LIN {X 0,Y 228.351,Z 344.664,A -85,B 0,C 180,E1 -20167.071,E2 -20167.071} C_VEL
LIN {X 0,Y 228.165,Z 344.686,A -85,B 0,C 180,E1 -20170.65,E2 -20170.65} C_VEL
LIN {X 0,Y 228.051,Z 344.704,A -85,B 0,C 180,E1 -20176.102,E2 -20176.102} C_VEL
LIN {X 0,Y 227.936,Z 344.714,A -85,B 0,C 180,E1 -20179.826,E2 -20179.826} C_VEL
LIN {X 0,Y 227.907,Z 344.72,A -85,B 0,C 180,E1 -20183.633,E2 -20183.633} C_VEL
LIN {X 0,Y 227.879,Z 344.721,A -85,B 0,C 180,E1 -20187.556,E2 -20187.556} C_VEL
LIN {X 0,Y 227.867,Z 344.726,A -85,B 0,C 180,E1 -20191.622,E2 -20191.622} C_VEL
LIN {X 0,Y 227.974,Z 344.855,A -85,B 0,C 180,E1 -20194.37,E2 -20194.37} C_VEL
LIN {X 0,Y 229.283,Z 351.773,A -85,B 0,C 180,E1 -20198.929,E2 -20198.929} C_VEL
LIN {X 0,Y 231.078,Z 360.512,A -85,B 0,C 180,E1 -20204.388,E2 -20204.388} C_VEL
LIN {X 0,Y 232.42,Z 367.069,A -85,B 0,C 180,E1 -20208.302,E2 -20208.302} C_VEL
LIN {X 0,Y 231.376,Z 372.602,A -85,B 0,C 180,E1 -20211.43,E2 -20211.43} C_VEL
LIN {X 0,Y 229.532,Z 381.682,A -85,B 0,C 180,E1 -20216.557,E2 -20216.557} C_VEL
LIN {X 0,Y 228.619,Z 387.309,A -85,B 0,C 180,E1 -20219.581,E2 -20219.581} C_VEL
LIN {X 0,Y 229.454,Z 407.428,A -85,B 0,C 180,E1 -20221.235,E2 -20221.235} C_VEL
LIN {X 0,Y 229.647,Z 410.827,A -85,B 0,C 180,E1 -20221.565,E2 -20221.565} C_VEL
LIN {X 0,Y 229.388,Z 416.398,A -85,B 0,C 180,E1 -20222.127,E2 -20222.127} C_VEL
LIN {X 0,Y 226.978,Z 425.249,A -85,B 0,C 180,E1 -20223.098,E2 -20223.098} C_VEL
LIN {X 0,Y 224.51,Z 433.801,A -85,B 0,C 180,E1 -20224.199,E2 -20224.199} C_VEL
LIN {X 0,Y 224.14,Z 438.823,A -85,B 0,C 180,E1 -20224.956,E2 -20224.956} C_VEL
LIN {X 0,Y 225.046,Z 452.21,A -85,B 0,C 180,E1 -20227.268,E2 -20227.268} C_VEL
LIN {X 0,Y 225.004,Z 455.94,A -85,B 0,C 180,E1 -20227.989,E2 -20227.989} C_VEL
LIN {X 0,Y 223.355,Z 467.739,A -85,B 0,C 180,E1 -20230.632,E2 -20230.632} C_VEL
LIN {X 0,Y 221.995,Z 477.991,A -85,B 0,C 180,E1 -20233.447,E2 -20233.447} C_VEL
LIN {X 0,Y 221.257,Z 486.356,A -85,B 0,C 180,E1 -20236.22,E2 -20236.22} C_VEL
LIN {X 0,Y 221.057,Z 493.355,A -85,B 0,C 180,E1 -20239.005,E2 -20239.005} C_VEL
LIN {X 0,Y 221.203,Z 499.088,A -85,B 0,C 180,E1 -20241.782,E2 -20241.782} C_VEL
LIN {X 0,Y 221.557,Z 503.69,A -85,B 0,C 180,E1 -20244.541,E2 -20244.541} C_VEL
LIN {X 0,Y 221.876,Z 506.14,A -85,B 0,C 180,E1 -20246.37,E2 -20246.37} C_VEL
LIN {X 0,Y 222.107,Z 508.099,A -85,B 0,C 180,E1 -20248.188,E2 -20248.188} C_VEL
LIN {X 0,Y 222.354,Z 509.63,A -85,B 0,C 180,E1 -20250.002,E2 -20250.002} C_VEL
LIN {X 0,Y 221.73,Z 510.553,A -85,B 0,C 180,E1 -20251.818,E2 -20251.818} C_VEL
LIN {X 0,Y 220.533,Z 511.308,A -85,B 0,C 180,E1 -20255.488,E2 -20255.488} C_VEL
LIN {X 0,Y 219.744,Z 510.766,A -85,B 0,C 180,E1 -20259.203,E2 -20259.203} C_VEL
LIN {X 0,Y 219.781,Z 509.022,A -85,B 0,C 180,E1 -20262.936,E2 -20262.936} C_VEL
LIN {X 0,Y 220.864,Z 506.171,A -85,B 0,C 180,E1 -20266.643,E2 -20266.643} C_VEL
LIN {X 0,Y 223.015,Z 502.256,A -85,B 0,C 180,E1 -20270.284,E2 -20270.284} C_VEL
LIN {X 0,Y 226.28,Z 497.299,A -85,B 0,C 180,E1 -20273.815,E2 -20273.815} C_VEL
LIN {X 0,Y 232.087,Z 489.566,A -85,B 0,C 180,E1 -20277.995,E2 -20277.995} C_VEL
LIN {X 0,Y 237.04,Z 483.14,A -85,B 0,C 180,E1 -20280.762,E2 -20280.762} C_VEL
LIN {X 0,Y 242.014,Z 476.891,A -85,B 0,C 180,E1 -20282.992,E2 -20282.992} C_VEL
LIN {X 0,Y 249.318,Z 466.525,A -85,B 0,C 180,E1 -20286.298,E2 -20286.298} C_VEL
LIN {X 0,Y 253.481,Z 460.309,A -85,B 0,C 180,E1 -20288.092,E2 -20288.092} C_VEL
LIN {X 0,Y 258.603,Z 451.554,A -85,B 0,C 180,E1 -20290.712,E2 -20290.712} C_VEL
LIN {X 0,Y 262.82,Z 443.829,A -85,B 0,C 180,E1 -20293.242,E2 -20293.242} C_VEL
LIN {X 0,Y 267.388,Z 435.806,A -85,B 0,C 180,E1 -20296.26,E2 -20296.26} C_VEL
LIN {X 0,Y 268.712,Z 433.696,A -85,B 0,C 180,E1 -20297.156,E2 -20297.156} C_VEL
LIN {X 0,Y 269.675,Z 431.962,A -85,B 0,C 180,E1 -20298.28,E2 -20298.28} C_VEL
LIN {X 0,Y 270.402,Z 430.463,A -85,B 0,C 180,E1 -20301.407,E2 -20301.407} C_VEL
LIN {X 0,Y 270.864,Z 430.408,A -85,B 0,C 180,E1 -20303.549,E2 -20303.549} C_VEL
LIN {X 0,Y 270.034,Z 431.543,A -85,B 0,C 180,E1 -20304.344,E2 -20304.344} C_VEL
LIN {X 0,Y 260.6,Z 440.793,A -85,B 0,C 180,E1 -20307.36,E2 -20307.36} C_VEL
LIN {X 0,Y 253.365,Z 447.035,A -85,B 0,C 180,E1 -20310.047,E2 -20310.047} C_VEL
LIN {X 0,Y 246.809,Z 451.946,A -85,B 0,C 180,E1 -20312.896,E2 -20312.896} C_VEL
LIN {X 0,Y 241.057,Z 455.609,A -85,B 0,C 180,E1 -20315.91,E2 -20315.91} C_VEL
LIN {X 0,Y 235.987,Z 458.133,A -85,B 0,C 180,E1 -20319.061,E2 -20319.061} C_VEL
LIN {X 0,Y 231.716,Z 459.508,A -85,B 0,C 180,E1 -20322.344,E2 -20322.344} C_VEL
LIN {X 0,Y 228.11,Z 459.778,A -85,B 0,C 180,E1 -20325.731,E2 -20325.731} C_VEL
LIN {X 0,Y 225.275,Z 458.892,A -85,B 0,C 180,E1 -20329.212,E2 -20329.212} C_VEL
LIN {X 0,Y 223.148,Z 456.815,A -85,B 0,C 180,E1 -20332.763,E2 -20332.763} C_VEL
LIN {X 0,Y 221.835,Z 453.504,A -85,B 0,C 180,E1 -20336.368,E2 -20336.368} C_VEL
LIN {X 0,Y 221.174,Z 448.92,A -85,B 0,C 180,E1 -20340,E2 -20340} C_VEL
LIN {X 0,Y 220.811,Z 442.957,A -85,B 0,C 180,E1 -20343.65,E2 -20343.65} C_VEL
LIN {X 0,Y 221.237,Z 435.436,A -85,B 0,C 180,E1 -20347.301,E2 -20347.301} C_VEL
LIN {X 0,Y 222.005,Z 427.386,A -85,B 0,C 180,E1 -20350.488,E2 -20350.488} C_VEL
LIN {X 0,Y 223.089,Z 417.659,A -85,B 0,C 180,E1 -20353.667,E2 -20353.667} C_VEL
LIN {X 0,Y 224.375,Z 407.773,A -85,B 0,C 180,E1 -20356.374,E2 -20356.374} C_VEL
LIN {X 0,Y 226.11,Z 394.99,A -85,B 0,C 180,E1 -20359.284,E2 -20359.284} C_VEL
LIN {X 0,Y 228.029,Z 382.007,A -85,B 0,C 180,E1 -20361.707,E2 -20361.707} C_VEL
LIN {X 0,Y 228.741,Z 375.181,A -85,B 0,C 180,E1 -20362.815,E2 -20362.815} C_VEL
LIN {X 0,Y 224.992,Z 361.192,A -85,B 0,C 180,E1 -20365.058,E2 -20365.058} C_VEL
LIN {X 0,Y 220.994,Z 346.136,A -85,B 0,C 180,E1 -20367.173,E2 -20367.173} C_VEL
LIN {X 0,Y 220.946,Z 345.626,A -85,B 0,C 180,E1 -20367.474,E2 -20367.474} C_VEL
LIN {X 0,Y 220.869,Z 345.599,A -85,B 0,C 180,E1 -20370.778,E2 -20370.778} C_VEL
LIN {X 0,Y 220.807,Z 345.604,A -85,B 0,C 180,E1 -20374.955,E2 -20374.955} C_VEL
LIN {X 0,Y 220.812,Z 345.602,A -85,B 0,C 180,E1 -20379.536,E2 -20379.536} C_VEL
LIN {X 0,Y 220.781,Z 345.607,A -85,B 0,C 180,E1 -20384.453,E2 -20384.453} C_VEL
LIN {X 0,Y 220.809,Z 345.604,A -85,B 0,C 180,E1 -20388.055,E2 -20388.055} C_VEL
LIN {X 0,Y 220.84,Z 345.597,A -85,B 0,C 180,E1 -20392.794,E2 -20392.794} C_VEL
LIN {X 0,Y 220.829,Z 345.601,A -85,B 0,C 180,E1 -20397.244,E2 -20397.244} C_VEL
LIN {X 0,Y 220.833,Z 345.598,A -85,B 0,C 180,E1 -20401.484,E2 -20401.484} C_VEL
LIN {X 0,Y 220.868,Z 345.596,A -85,B 0,C 180,E1 -20405.563,E2 -20405.563} C_VEL
LIN {X 0,Y 220.891,Z 345.592,A -85,B 0,C 180,E1 -20409.512,E2 -20409.512} C_VEL
LIN {X 0,Y 221.022,Z 345.576,A -85,B 0,C 180,E1 -20413.369,E2 -20413.369} C_VEL
LIN {X 0,Y 221.122,Z 345.561,A -85,B 0,C 180,E1 -20419.005,E2 -20419.005} C_VEL
LIN {X 0,Y 221.316,Z 345.54,A -85,B 0,C 180,E1 -20422.701,E2 -20422.701} C_VEL
LIN {X 0,Y 221.517,Z 345.514,A -85,B 0,C 180,E1 -20428.18,E2 -20428.18} C_VEL
LIN {X 0,Y 221.517,Z 345.518,A -85,B 0,C 180,E1 -20431.816,E2 -20431.816} C_VEL
LIN {X 0,Y 221.315,Z 345.539,A -85,B 0,C 180,E1 -20437.296,E2 -20437.296} C_VEL
LIN {X 0,Y 221.12,Z 345.565,A -85,B 0,C 180,E1 -20440.992,E2 -20440.992} C_VEL
LIN {X 0,Y 221.019,Z 345.576,A -85,B 0,C 180,E1 -20446.628,E2 -20446.628} C_VEL
LIN {X 0,Y 220.894,Z 345.592,A -85,B 0,C 180,E1 -20450.484,E2 -20450.484} C_VEL
LIN {X 0,Y 220.868,Z 345.593,A -85,B 0,C 180,E1 -20454.433,E2 -20454.433} C_VEL
LIN {X 0,Y 220.827,Z 345.601,A -85,B 0,C 180,E1 -20458.513,E2 -20458.513} C_VEL
LIN {X 0,Y 220.815,Z 345.6,A -85,B 0,C 180,E1 -20462.754,E2 -20462.754} C_VEL
LIN {X 0,Y 220.808,Z 345.606,A -85,B 0,C 180,E1 -20467.276,E2 -20467.276} C_VEL
LIN {X 0,Y 220.768,Z 345.607,A -85,B 0,C 180,E1 -20471.95,E2 -20471.95} C_VEL
LIN {X 0,Y 220.772,Z 345.609,A -85,B 0,C 180,E1 -20475.545,E2 -20475.545} C_VEL
LIN {X 0,Y 220.803,Z 345.602,A -85,B 0,C 180,E1 -20480.461,E2 -20480.461} C_VEL
LIN {X 0,Y 220.796,Z 345.607,A -85,B 0,C 180,E1 -20485.043,E2 -20485.043} C_VEL
LIN {X 0,Y 220.863,Z 345.596,A -85,B 0,C 180,E1 -20489.393,E2 -20489.393} C_VEL
LIN {X 0,Y 220.89,Z 345.593,A -85,B 0,C 180,E1 -20493.548,E2 -20493.548} C_VEL
LIN {X 0,Y 220.872,Z 345.594,A -85,B 0,C 180,E1 -20497.552,E2 -20497.552} C_VEL
LIN {X 0,Y 220.978,Z 345.585,A -85,B 0,C 180,E1 -20502.57,E2 -20502.57} C_VEL
LIN {X 0,Y 221.02,Z 345.577,A -85,B 0,C 180,E1 -20507.138,E2 -20507.138} C_VEL
LIN {X 0,Y 221.252,Z 345.549,A -85,B 0,C 180,E1 -20510.861,E2 -20510.861} C_VEL
LIN {X 0,Y 221.305,Z 345.54,A -85,B 0,C 180,E1 -20512.702,E2 -20512.702} C_VEL
LIN {X 0,Y 221.507,Z 345.519,A -85,B 0,C 180,E1 -20518.181,E2 -20518.181} C_VEL
LIN {X 0,Y 221.507,Z 345.514,A -85,B 0,C 180,E1 -20521.818,E2 -20521.818} C_VEL
LIN {X 0,Y 221.304,Z 345.541,A -85,B 0,C 180,E1 -20527.297,E2 -20527.297} C_VEL
LIN {X 0,Y 221.11,Z 345.563,A -85,B 0,C 180,E1 -20530.994,E2 -20530.994} C_VEL
LIN {X 0,Y 221.01,Z 345.578,A -85,B 0,C 180,E1 -20536.63,E2 -20536.63} C_VEL
LIN {X 0,Y 220.886,Z 345.594,A -85,B 0,C 180,E1 -20540.486,E2 -20540.486} C_VEL
LIN {X 0,Y 220.86,Z 345.598,A -85,B 0,C 180,E1 -20544.435,E2 -20544.435} C_VEL
LIN {X 0,Y 220.829,Z 345.6,A -85,B 0,C 180,E1 -20548.514,E2 -20548.514} C_VEL
LIN {X 0,Y 220.837,Z 345.602,A -85,B 0,C 180,E1 -20552.752,E2 -20552.752} C_VEL
LIN {X 0,Y 220.932,Z 345.761,A -85,B 0,C 180,E1 -20554.204,E2 -20554.204} C_VEL
LIN {X 0,Y 222.336,Z 353.162,A -85,B 0,C 180,E1 -20559.212,E2 -20559.212} C_VEL
LIN {X 0,Y 223.801,Z 360.205,A -85,B 0,C 180,E1 -20563.761,E2 -20563.761} C_VEL
LIN {X 0,Y 225.071,Z 366.093,A -85,B 0,C 180,E1 -20567.402,E2 -20567.402} C_VEL
LIN {X 0,Y 225.155,Z 368.839,A -85,B 0,C 180,E1 -20569.045,E2 -20569.045} C_VEL
LIN {X 0,Y 223.522,Z 376.147,A -85,B 0,C 180,E1 -20573.318,E2 -20573.318} C_VEL
LIN {X 0,Y 221.784,Z 385.568,A -85,B 0,C 180,E1 -20578.824,E2 -20578.824} C_VEL
LIN {X 0,Y 221.637,Z 386.569,A -85,B 0,C 180,E1 -20579.183,E2 -20579.183} C_VEL
LIN {X 0,Y 222.275,Z 404.267,A -85,B 0,C 180,E1 -20580.656,E2 -20580.656} C_VEL
LIN {X 0,Y 223.092,Z 419.696,A -85,B 0,C 180,E1 -20582.314,E2 -20582.314} C_VEL
LIN {X 0,Y 223.769,Z 433.244,A -85,B 0,C 180,E1 -20584.107,E2 -20584.107} C_VEL
LIN {X 0,Y 224.14,Z 438.823,A -85,B 0,C 180,E1 -20584.956,E2 -20584.956} C_VEL
LIN {X 0,Y 223.745,Z 443.842,A -85,B 0,C 180,E1 -20585.768,E2 -20585.768} C_VEL
LIN {X 0,Y 222.288,Z 448.619,A -85,B 0,C 180,E1 -20586.612,E2 -20586.612} C_VEL
LIN {X 0,Y 218.377,Z 457.615,A -85,B 0,C 180,E1 -20588.445,E2 -20588.445} C_VEL
LIN {X 0,Y 216.763,Z 463.504,A -85,B 0,C 180,E1 -20589.815,E2 -20589.815} C_VEL
LIN {X 0,Y 215.405,Z 473.343,A -85,B 0,C 180,E1 -20592.436,E2 -20592.436} C_VEL
LIN {X 0,Y 214.541,Z 482.269,A -85,B 0,C 180,E1 -20595.295,E2 -20595.295} C_VEL
LIN {X 0,Y 214.11,Z 490.839,A -85,B 0,C 180,E1 -20598.643,E2 -20598.643} C_VEL
LIN {X 0,Y 214.234,Z 496.795,A -85,B 0,C 180,E1 -20601.513,E2 -20601.513} C_VEL
LIN {X 0,Y 214.615,Z 501.559,A -85,B 0,C 180,E1 -20604.364,E2 -20604.364} C_VEL
LIN {X 0,Y 215.06,Z 505.244,A -85,B 0,C 180,E1 -20607.192,E2 -20607.192} C_VEL
LIN {X 0,Y 215.447,Z 507.895,A -85,B 0,C 180,E1 -20610.002,E2 -20610.002} C_VEL
LIN {X 0,Y 214.794,Z 508.897,A -85,B 0,C 180,E1 -20611.877,E2 -20611.877} C_VEL
LIN {X 0,Y 213.518,Z 509.799,A -85,B 0,C 180,E1 -20615.669,E2 -20615.669} C_VEL
LIN {X 0,Y 212.721,Z 509.42,A -85,B 0,C 180,E1 -20619.51,E2 -20619.51} C_VEL
LIN {X 0,Y 212.816,Z 507.904,A -85,B 0,C 180,E1 -20623.367,E2 -20623.367} C_VEL
LIN {X 0,Y 214.004,Z 505.324,A -85,B 0,C 180,E1 -20627.193,E2 -20627.193} C_VEL
LIN {X 0,Y 216.31,Z 501.701,A -85,B 0,C 180,E1 -20630.942,E2 -20630.942} C_VEL
LIN {X 0,Y 219.763,Z 497.027,A -85,B 0,C 180,E1 -20634.567,E2 -20634.567} C_VEL
LIN {X 0,Y 225.822,Z 489.776,A -85,B 0,C 180,E1 -20638.843,E2 -20638.843} C_VEL
LIN {X 0,Y 230.142,Z 484.601,A -85,B 0,C 180,E1 -20641.276,E2 -20641.276} C_VEL
LIN {X 0,Y 236.156,Z 477.821,A -85,B 0,C 180,E1 -20643.919,E2 -20643.919} C_VEL
LIN {X 0,Y 243.775,Z 468.048,A -85,B 0,C 180,E1 -20647.261,E2 -20647.261} C_VEL
LIN {X 0,Y 248.127,Z 462.176,A -85,B 0,C 180,E1 -20649.067,E2 -20649.067} C_VEL
LIN {X 0,Y 253.567,Z 453.945,A -85,B 0,C 180,E1 -20651.699,E2 -20651.699} C_VEL
LIN {X 0,Y 258.074,Z 446.707,A -85,B 0,C 180,E1 -20654.242,E2 -20654.242} C_VEL
LIN {X 0,Y 263.047,Z 439.181,A -85,B 0,C 180,E1 -20657.258,E2 -20657.258} C_VEL
LIN {X 0,Y 264.384,Z 437.174,A -85,B 0,C 180,E1 -20658.351,E2 -20658.351} C_VEL
LIN {X 0,Y 264.998,Z 435.771,A -85,B 0,C 180,E1 -20660.469,E2 -20660.469} C_VEL
LIN {X 0,Y 265.436,Z 435.247,A -85,B 0,C 180,E1 -20662.592,E2 -20662.592} C_VEL
LIN {X 0,Y 265.37,Z 435.437,A -85,B 0,C 180,E1 -20663.475,E2 -20663.475} C_VEL
LIN {X 0,Y 257.271,Z 442.713,A -85,B 0,C 180,E1 -20665.944,E2 -20665.944} C_VEL
LIN {X 0,Y 249.612,Z 448.804,A -85,B 0,C 180,E1 -20668.609,E2 -20668.609} C_VEL
LIN {X 0,Y 242.586,Z 453.632,A -85,B 0,C 180,E1 -20671.444,E2 -20671.444} C_VEL
LIN {X 0,Y 234.939,Z 457.918,A -85,B 0,C 180,E1 -20675.242,E2 -20675.242} C_VEL
LIN {X 0,Y 229.646,Z 460.108,A -85,B 0,C 180,E1 -20678.455,E2 -20678.455} C_VEL
LIN {X 0,Y 225.174,Z 461.172,A -85,B 0,C 180,E1 -20681.814,E2 -20681.814} C_VEL
LIN {X 0,Y 221.378,Z 461.155,A -85,B 0,C 180,E1 -20685.288,E2 -20685.288} C_VEL
LIN {X 0,Y 218.394,Z 459.99,A -85,B 0,C 180,E1 -20688.868,E2 -20688.868} C_VEL
LIN {X 0,Y 216.167,Z 457.648,A -85,B 0,C 180,E1 -20692.528,E2 -20692.528} C_VEL
LIN {X 0,Y 214.773,Z 454.086,A -85,B 0,C 180,E1 -20696.248,E2 -20696.248} C_VEL
LIN {X 0,Y 214.083,Z 449.252,A -85,B 0,C 180,E1 -20700,E2 -20700} C_VEL
LIN {X 0,Y 213.806,Z 444.714,A -85,B 0,C 180,E1 -20702.827,E2 -20702.827} C_VEL
LIN {X 0,Y 214.012,Z 437.308,A -85,B 0,C 180,E1 -20706.601,E2 -20706.601} C_VEL
LIN {X 0,Y 214.782,Z 429.439,A -85,B 0,C 180,E1 -20709.876,E2 -20709.876} C_VEL
LIN {X 0,Y 215.777,Z 419.916,A -85,B 0,C 180,E1 -20713.18,E2 -20713.18} C_VEL
LIN {X 0,Y 217.015,Z 410.235,A -85,B 0,C 180,E1 -20715.979,E2 -20715.979} C_VEL
LIN {X 0,Y 218.678,Z 397.716,A -85,B 0,C 180,E1 -20718.991,E2 -20718.991} C_VEL
LIN {X 0,Y 220.538,Z 385.108,A -85,B 0,C 180,E1 -20721.499,E2 -20721.499} C_VEL
LIN {X 0,Y 221.642,Z 377.103,A -85,B 0,C 180,E1 -20722.861,E2 -20722.861} C_VEL
LIN {X 0,Y 220.676,Z 372.535,A -85,B 0,C 180,E1 -20723.657,E2 -20723.657} C_VEL
LIN {X 0,Y 217.362,Z 359.912,A -85,B 0,C 180,E1 -20725.67,E2 -20725.67} C_VEL
LIN {X 0,Y 213.977,Z 347.004,A -85,B 0,C 180,E1 -20727.522,E2 -20727.522} C_VEL
LIN {X 0,Y 213.855,Z 346.502,A -85,B 0,C 180,E1 -20727.871,E2 -20727.871} C_VEL
LIN {X 0,Y 213.783,Z 346.48,A -85,B 0,C 180,E1 -20731.736,E2 -20731.736} C_VEL
LIN {X 0,Y 213.75,Z 346.484,A -85,B 0,C 180,E1 -20736.288,E2 -20736.288} C_VEL
LIN {X 0,Y 213.718,Z 346.487,A -85,B 0,C 180,E1 -20741.125,E2 -20741.125} C_VEL
LIN {X 0,Y 213.754,Z 346.482,A -85,B 0,C 180,E1 -20746.332,E2 -20746.332} C_VEL
LIN {X 0,Y 213.744,Z 346.483,A -85,B 0,C 180,E1 -20751.336,E2 -20751.336} C_VEL
LIN {X 0,Y 213.776,Z 346.48,A -85,B 0,C 180,E1 -20756.02,E2 -20756.02} C_VEL
LIN {X 0,Y 213.766,Z 346.48,A -85,B 0,C 180,E1 -20760.45,E2 -20760.45} C_VEL
LIN {X 0,Y 213.804,Z 346.476,A -85,B 0,C 180,E1 -20764.7,E2 -20764.7} C_VEL
LIN {X 0,Y 213.809,Z 346.474,A -85,B 0,C 180,E1 -20768.801,E2 -20768.801} C_VEL
LIN {X 0,Y 213.949,Z 346.457,A -85,B 0,C 180,E1 -20772.802,E2 -20772.802} C_VEL
LIN {X 0,Y 213.986,Z 346.453,A -85,B 0,C 180,E1 -20776.707,E2 -20776.707} C_VEL
LIN {X 0,Y 214.202,Z 346.425,A -85,B 0,C 180,E1 -20780.556,E2 -20780.556} C_VEL
LIN {X 0,Y 214.253,Z 346.42,A -85,B 0,C 180,E1 -20782.459,E2 -20782.459} C_VEL
LIN {X 0,Y 214.45,Z 346.394,A -85,B 0,C 180,E1 -20788.12,E2 -20788.12} C_VEL
LIN {X 0,Y 214.555,Z 346.384,A -85,B 0,C 180,E1 -20789.998,E2 -20789.998} C_VEL
LIN {X 0,Y 214.45,Z 346.398,A -85,B 0,C 180,E1 -20791.876,E2 -20791.876} C_VEL
LIN {X 0,Y 214.252,Z 346.42,A -85,B 0,C 180,E1 -20797.538,E2 -20797.538} C_VEL
LIN {X 0,Y 214.05,Z 346.448,A -85,B 0,C 180,E1 -20801.36,E2 -20801.36} C_VEL
LIN {X 0,Y 213.936,Z 346.458,A -85,B 0,C 180,E1 -20805.235,E2 -20805.235} C_VEL
LIN {X 0,Y 213.87,Z 346.47,A -85,B 0,C 180,E1 -20809.183,E2 -20809.183} C_VEL
LIN {X 0,Y 213.848,Z 346.47,A -85,B 0,C 180,E1 -20813.225,E2 -20813.225} C_VEL
LIN {X 0,Y 213.829,Z 346.476,A -85,B 0,C 180,E1 -20817.448,E2 -20817.448} C_VEL
LIN {X 0,Y 213.767,Z 346.478,A -85,B 0,C 180,E1 -20821.735,E2 -20821.735} C_VEL
LIN {X 0,Y 213.742,Z 346.484,A -85,B 0,C 180,E1 -20826.286,E2 -20826.286} C_VEL
LIN {X 0,Y 213.71,Z 346.487,A -85,B 0,C 180,E1 -20831.123,E2 -20831.123} C_VEL
LIN {X 0,Y 213.705,Z 346.489,A -85,B 0,C 180,E1 -20833.676,E2 -20833.676} C_VEL
LIN {X 0,Y 213.704,Z 346.488,A -85,B 0,C 180,E1 -20836.342,E2 -20836.342} C_VEL
LIN {X 0,Y 213.714,Z 346.487,A -85,B 0,C 180,E1 -20839.141,E2 -20839.141} C_VEL
LIN {X 0,Y 213.739,Z 346.484,A -85,B 0,C 180,E1 -20843.71,E2 -20843.71} C_VEL
LIN {X 0,Y 213.79,Z 346.477,A -85,B 0,C 180,E1 -20848.723,E2 -20848.723} C_VEL
LIN {X 0,Y 213.821,Z 346.476,A -85,B 0,C 180,E1 -20852.602,E2 -20852.602} C_VEL
LIN {X 0,Y 213.847,Z 346.471,A -85,B 0,C 180,E1 -20856.951,E2 -20856.951} C_VEL
LIN {X 0,Y 213.927,Z 346.462,A -85,B 0,C 180,E1 -20862.304,E2 -20862.304} C_VEL
LIN {X 0,Y 213.974,Z 346.457,A -85,B 0,C 180,E1 -20866.707,E2 -20866.707} C_VEL
LIN {X 0,Y 214.19,Z 346.43,A -85,B 0,C 180,E1 -20870.557,E2 -20870.557} C_VEL
LIN {X 0,Y 214.242,Z 346.421,A -85,B 0,C 180,E1 -20872.46,E2 -20872.46} C_VEL
LIN {X 0,Y 214.44,Z 346.399,A -85,B 0,C 180,E1 -20878.121,E2 -20878.121} C_VEL
LIN {X 0,Y 214.544,Z 346.385,A -85,B 0,C 180,E1 -20880,E2 -20880} C_VEL
LIN {X 0,Y 214.44,Z 346.395,A -85,B 0,C 180,E1 -20881.878,E2 -20881.878} C_VEL
LIN {X 0,Y 214.241,Z 346.421,A -85,B 0,C 180,E1 -20887.539,E2 -20887.539} C_VEL
LIN {X 0,Y 214.041,Z 346.444,A -85,B 0,C 180,E1 -20891.362,E2 -20891.362} C_VEL
LIN {X 0,Y 213.927,Z 346.461,A -85,B 0,C 180,E1 -20895.237,E2 -20895.237} C_VEL
LIN {X 0,Y 213.833,Z 346.468,A -85,B 0,C 180,E1 -20899.188,E2 -20899.188} C_VEL
LIN {X 0,Y 213.84,Z 346.471,A -85,B 0,C 180,E1 -20903.227,E2 -20903.227} C_VEL
LIN {X 0,Y 213.822,Z 346.471,A -85,B 0,C 180,E1 -20907.45,E2 -20907.45} C_VEL
LIN {X 0,Y 213.795,Z 346.479,A -85,B 0,C 180,E1 -20912.847,E2 -20912.847} C_VEL
LIN {X 0,Y 213.868,Z 346.565,A -85,B 0,C 180,E1 -20913.962,E2 -20913.962} C_VEL
LIN {X 0,Y 215.074,Z 352.823,A -85,B 0,C 180,E1 -20918.379,E2 -20918.379} C_VEL
LIN {X 0,Y 216.736,Z 360.905,A -85,B 0,C 180,E1 -20923.769,E2 -20923.769} C_VEL
LIN {X 0,Y 218.058,Z 367.282,A -85,B 0,C 180,E1 -20927.841,E2 -20927.841} C_VEL
LIN {X 0,Y 218.085,Z 368.957,A -85,B 0,C 180,E1 -20928.868,E2 -20928.868} C_VEL
LIN {X 0,Y 216.473,Z 375.913,A -85,B 0,C 180,E1 -20933.088,E2 -20933.088} C_VEL
LIN {X 0,Y 214.757,Z 385.006,A -85,B 0,C 180,E1 -20938.565,E2 -20938.565} C_VEL
LIN {X 0,Y 214.689,Z 385.675,A -85,B 0,C 180,E1 -20938.76,E2 -20938.76} C_VEL
LIN {X 0,Y 215.195,Z 403.156,A -85,B 0,C 180,E1 -20940.266,E2 -20940.266} C_VEL
LIN {X 0,Y 216.002,Z 419.204,A -85,B 0,C 180,E1 -20942.062,E2 -20942.062} C_VEL
LIN {X 0,Y 216.637,Z 432.147,A -85,B 0,C 180,E1 -20943.847,E2 -20943.847} C_VEL
LIN {X 0,Y 217.538,Z 446.165,A -85,B 0,C 180,E1 -20946.184,E2 -20946.184} C_VEL
LIN {X 0,Y 218.079,Z 454.299,A -85,B 0,C 180,E1 -20947.751,E2 -20947.751} C_VEL
LIN {X 0,Y 216.763,Z 463.504,A -85,B 0,C 180,E1 -20949.815,E2 -20949.815} C_VEL
LIN {X 0,Y 216.117,Z 466.329,A -85,B 0,C 180,E1 -20950.522,E2 -20950.522} C_VEL
LIN {X 0,Y 213.503,Z 471.438,A -85,B 0,C 180,E1 -20951.975,E2 -20951.975} C_VEL
LIN {X 0,Y 208.345,Z 479.394,A -85,B 0,C 180,E1 -20954.757,E2 -20954.757} C_VEL
LIN {X 0,Y 207.415,Z 482.803,A -85,B 0,C 180,E1 -20956.074,E2 -20956.074} C_VEL
LIN {X 0,Y 207.213,Z 491.125,A -85,B 0,C 180,E1 -20959.603,E2 -20959.603} C_VEL
LIN {X 0,Y 207.532,Z 497.838,A -85,B 0,C 180,E1 -20963.195,E2 -20963.195} C_VEL
LIN {X 0,Y 208.017,Z 502.084,A -85,B 0,C 180,E1 -20966.127,E2 -20966.127} C_VEL
LIN {X 0,Y 208.313,Z 504.301,A -85,B 0,C 180,E1 -20968.068,E2 -20968.068} C_VEL
LIN {X 0,Y 208.561,Z 506.058,A -85,B 0,C 180,E1 -20970.002,E2 -20970.002} C_VEL
LIN {X 0,Y 207.885,Z 507.149,A -85,B 0,C 180,E1 -20971.939,E2 -20971.939} C_VEL
LIN {X 0,Y 206.542,Z 508.233,A -85,B 0,C 180,E1 -20975.861,E2 -20975.861} C_VEL
LIN {X 0,Y 205.7,Z 508.058,A -85,B 0,C 180,E1 -20979.838,E2 -20979.838} C_VEL
LIN {X 0,Y 205.844,Z 506.771,A -85,B 0,C 180,E1 -20983.829,E2 -20983.829} C_VEL
LIN {X 0,Y 207.482,Z 503.899,A -85,B 0,C 180,E1 -20988.48,E2 -20988.48} C_VEL
LIN {X 0,Y 211.308,Z 498.999,A -85,B 0,C 180,E1 -20993.525,E2 -20993.525} C_VEL
LIN {X 0,Y 215.682,Z 494.188,A -85,B 0,C 180,E1 -20997.143,E2 -20997.143} C_VEL
LIN {X 0,Y 222.265,Z 487.043,A -85,B 0,C 180,E1 -21001.25,E2 -21001.25} C_VEL
LIN {X 0,Y 229.475,Z 479.619,A -85,B 0,C 180,E1 -21004.514,E2 -21004.514} C_VEL
LIN {X 0,Y 238.291,Z 469.453,A -85,B 0,C 180,E1 -21008.271,E2 -21008.271} C_VEL
LIN {X 0,Y 242.846,Z 463.939,A -85,B 0,C 180,E1 -21010.086,E2 -21010.086} C_VEL
LIN {X 0,Y 248.571,Z 456.237,A -85,B 0,C 180,E1 -21012.733,E2 -21012.733} C_VEL
LIN {X 0,Y 252.751,Z 450.352,A -85,B 0,C 180,E1 -21014.929,E2 -21014.929} C_VEL
LIN {X 0,Y 258.202,Z 443.029,A -85,B 0,C 180,E1 -21018.025,E2 -21018.025} C_VEL
LIN {X 0,Y 258.947,Z 442.032,A -85,B 0,C 180,E1 -21018.571,E2 -21018.571} C_VEL
LIN {X 0,Y 259.358,Z 441.24,A -85,B 0,C 180,E1 -21019.433,E2 -21019.433} C_VEL
LIN {X 0,Y 260.084,Z 439.935,A -85,B 0,C 180,E1 -21022.54,E2 -21022.54} C_VEL
LIN {X 0,Y 258.475,Z 441.282,A -85,B 0,C 180,E1 -21023.26,E2 -21023.26} C_VEL
LIN {X 0,Y 250.051,Z 447.869,A -85,B 0,C 180,E1 -21025.798,E2 -21025.798} C_VEL
LIN {X 0,Y 242.227,Z 453.192,A -85,B 0,C 180,E1 -21028.517,E2 -21028.517} C_VEL
LIN {X 0,Y 235.157,Z 457.278,A -85,B 0,C 180,E1 -21031.434,E2 -21031.434} C_VEL
LIN {X 0,Y 228.879,Z 460.222,A -85,B 0,C 180,E1 -21034.54,E2 -21034.54} C_VEL
LIN {X 0,Y 223.318,Z 462.084,A -85,B 0,C 180,E1 -21037.812,E2 -21037.812} C_VEL
LIN {X 0,Y 218.639,Z 462.836,A -85,B 0,C 180,E1 -21041.25,E2 -21041.25} C_VEL
LIN {X 0,Y 214.653,Z 462.524,A -85,B 0,C 180,E1 -21044.816,E2 -21044.816} C_VEL
LIN {X 0,Y 211.52,Z 461.072,A -85,B 0,C 180,E1 -21048.501,E2 -21048.501} C_VEL
LIN {X 0,Y 209.19,Z 458.453,A -85,B 0,C 180,E1 -21052.277,E2 -21052.277} C_VEL
LIN {X 0,Y 207.709,Z 454.623,A -85,B 0,C 180,E1 -21056.12,E2 -21056.12} C_VEL
LIN {X 0,Y 206.988,Z 449.505,A -85,B 0,C 180,E1 -21060.001,E2 -21060.001} C_VEL
LIN {X 0,Y 206.719,Z 444.754,A -85,B 0,C 180,E1 -21062.924,E2 -21062.924} C_VEL
LIN {X 0,Y 206.939,Z 437.077,A -85,B 0,C 180,E1 -21066.827,E2 -21066.827} C_VEL
LIN {X 0,Y 207.776,Z 428.379,A -85,B 0,C 180,E1 -21070.41,E2 -21070.41} C_VEL
LIN {X 0,Y 208.821,Z 419.016,A -85,B 0,C 180,E1 -21073.627,E2 -21073.627} C_VEL
LIN {X 0,Y 210.134,Z 409.008,A -85,B 0,C 180,E1 -21076.517,E2 -21076.517} C_VEL
LIN {X 0,Y 211.749,Z 397.205,A -85,B 0,C 180,E1 -21079.385,E2 -21079.385} C_VEL
LIN {X 0,Y 213.704,Z 384.294,A -85,B 0,C 180,E1 -21081.968,E2 -21081.968} C_VEL
LIN {X 0,Y 214.626,Z 377.52,A -85,B 0,C 180,E1 -21083.138,E2 -21083.138} C_VEL
LIN {X 0,Y 211.089,Z 363.812,A -85,B 0,C 180,E1 -21085.485,E2 -21085.485} C_VEL
LIN {X 0,Y 207.719,Z 351.017,A -85,B 0,C 180,E1 -21087.378,E2 -21087.378} C_VEL
LIN {X 0,Y 206.895,Z 347.841,A -85,B 0,C 180,E1 -21087.888,E2 -21087.888} C_VEL
LIN {X 0,Y 206.791,Z 347.353,A -85,B 0,C 180,E1 -21088.413,E2 -21088.413} C_VEL
LIN {X 0,Y 206.708,Z 347.362,A -85,B 0,C 180,E1 -21092.957,E2 -21092.957} C_VEL
LIN {X 0,Y 206.686,Z 347.36,A -85,B 0,C 180,E1 -21097.739,E2 -21097.739} C_VEL
LIN {X 0,Y 206.648,Z 347.367,A -85,B 0,C 180,E1 -21101.562,E2 -21101.562} C_VEL
LIN {X 0,Y 206.665,Z 347.361,A -85,B 0,C 180,E1 -21105.574,E2 -21105.574} C_VEL
LIN {X 0,Y 206.682,Z 347.364,A -85,B 0,C 180,E1 -21109.752,E2 -21109.752} C_VEL
LIN {X 0,Y 206.737,Z 347.356,A -85,B 0,C 180,E1 -21114.694,E2 -21114.694} C_VEL
LIN {X 0,Y 206.713,Z 347.359,A -85,B 0,C 180,E1 -21119.336,E2 -21119.336} C_VEL
LIN {X 0,Y 206.737,Z 347.355,A -85,B 0,C 180,E1 -21123.771,E2 -21123.771} C_VEL
LIN {X 0,Y 206.745,Z 347.358,A -85,B 0,C 180,E1 -21128.04,E2 -21128.04} C_VEL
LIN {X 0,Y 206.879,Z 347.34,A -85,B 0,C 180,E1 -21132.195,E2 -21132.195} C_VEL
LIN {X 0,Y 206.92,Z 347.335,A -85,B 0,C 180,E1 -21136.244,E2 -21136.244} C_VEL
LIN {X 0,Y 207.138,Z 347.306,A -85,B 0,C 180,E1 -21140.231,E2 -21140.231} C_VEL
LIN {X 0,Y 207.194,Z 347.301,A -85,B 0,C 180,E1 -21142.2,E2 -21142.2} C_VEL
LIN {X 0,Y 207.387,Z 347.275,A -85,B 0,C 180,E1 -21148.056,E2 -21148.056} C_VEL
LIN {X 0,Y 207.52,Z 347.26,A -85,B 0,C 180,E1 -21149.998,E2 -21149.998} C_VEL
LIN {X 0,Y 207.387,Z 347.277,A -85,B 0,C 180,E1 -21151.94,E2 -21151.94} C_VEL
LIN {X 0,Y 207.192,Z 347.301,A -85,B 0,C 180,E1 -21157.796,E2 -21157.796} C_VEL
LIN {X 0,Y 206.986,Z 347.327,A -85,B 0,C 180,E1 -21161.753,E2 -21161.753} C_VEL
LIN {X 0,Y 206.87,Z 347.34,A -85,B 0,C 180,E1 -21165.769,E2 -21165.769} C_VEL
LIN {X 0,Y 206.801,Z 347.349,A -85,B 0,C 180,E1 -21169.865,E2 -21169.865} C_VEL
LIN {X 0,Y 206.764,Z 347.35,A -85,B 0,C 180,E1 -21174.07,E2 -21174.07} C_VEL
LIN {X 0,Y 206.737,Z 347.356,A -85,B 0,C 180,E1 -21178.418,E2 -21178.418} C_VEL
LIN {X 0,Y 206.697,Z 347.359,A -85,B 0,C 180,E1 -21182.955,E2 -21182.955} C_VEL
LIN {X 0,Y 206.678,Z 347.364,A -85,B 0,C 180,E1 -21187.738,E2 -21187.738} C_VEL
LIN {X 0,Y 206.64,Z 347.368,A -85,B 0,C 180,E1 -21191.561,E2 -21191.561} C_VEL
LIN {X 0,Y 206.631,Z 347.37,A -85,B 0,C 180,E1 -21195.579,E2 -21195.579} C_VEL
LIN {X 0,Y 206.657,Z 347.364,A -85,B 0,C 180,E1 -21199.747,E2 -21199.747} C_VEL
LIN {X 0,Y 206.695,Z 347.364,A -85,B 0,C 180,E1 -21204.687,E2 -21204.687} C_VEL
LIN {X 0,Y 206.719,Z 347.358,A -85,B 0,C 180,E1 -21209.338,E2 -21209.338} C_VEL
LIN {X 0,Y 206.728,Z 347.357,A -85,B 0,C 180,E1 -21213.771,E2 -21213.771} C_VEL
LIN {X 0,Y 206.752,Z 347.353,A -85,B 0,C 180,E1 -21218.042,E2 -21218.042} C_VEL
LIN {X 0,Y 206.871,Z 347.34,A -85,B 0,C 180,E1 -21222.196,E2 -21222.196} C_VEL
LIN {X 0,Y 206.908,Z 347.334,A -85,B 0,C 180,E1 -21226.245,E2 -21226.245} C_VEL
LIN {X 0,Y 207.127,Z 347.31,A -85,B 0,C 180,E1 -21230.232,E2 -21230.232} C_VEL
LIN {X 0,Y 207.182,Z 347.301,A -85,B 0,C 180,E1 -21232.201,E2 -21232.201} C_VEL
LIN {X 0,Y 207.377,Z 347.278,A -85,B 0,C 180,E1 -21238.057,E2 -21238.057} C_VEL
LIN {X 0,Y 207.508,Z 347.261,A -85,B 0,C 180,E1 -21239.999,E2 -21239.999} C_VEL
LIN {X 0,Y 207.377,Z 347.275,A -85,B 0,C 180,E1 -21241.942,E2 -21241.942} C_VEL
LIN {X 0,Y 207.182,Z 347.302,A -85,B 0,C 180,E1 -21247.798,E2 -21247.798} C_VEL
LIN {X 0,Y 206.976,Z 347.325,A -85,B 0,C 180,E1 -21251.755,E2 -21251.755} C_VEL
LIN {X 0,Y 206.86,Z 347.342,A -85,B 0,C 180,E1 -21255.771,E2 -21255.771} C_VEL
LIN {X 0,Y 206.777,Z 347.349,A -85,B 0,C 180,E1 -21259.869,E2 -21259.869} C_VEL
LIN {X 0,Y 206.757,Z 347.356,A -85,B 0,C 180,E1 -21264.073,E2 -21264.073} C_VEL
LIN {X 0,Y 206.737,Z 347.355,A -85,B 0,C 180,E1 -21268.419,E2 -21268.419} C_VEL
LIN {X 0,Y 206.845,Z 347.42,A -85,B 0,C 180,E1 -21273.805,E2 -21273.805} C_VEL
LIN {X 0,Y 208.22,Z 354.703,A -85,B 0,C 180,E1 -21279.079,E2 -21279.079} C_VEL
LIN {X 0,Y 209.532,Z 361.05,A -85,B 0,C 180,E1 -21283.438,E2 -21283.438} C_VEL
LIN {X 0,Y 210.815,Z 366.672,A -85,B 0,C 180,E1 -21287.173,E2 -21287.173} C_VEL
LIN {X 0,Y 210.807,Z 370.007,A -85,B 0,C 180,E1 -21289.301,E2 -21289.301} C_VEL
LIN {X 0,Y 208.883,Z 378.126,A -85,B 0,C 180,E1 -21294.426,E2 -21294.426} C_VEL
LIN {X 0,Y 207.761,Z 384.279,A -85,B 0,C 180,E1 -21298.237,E2 -21298.237} C_VEL
LIN {X 0,Y 207.689,Z 388.874,A -85,B 0,C 180,E1 -21298.687,E2 -21298.687} C_VEL
LIN {X 0,Y 208.174,Z 403.78,A -85,B 0,C 180,E1 -21300.06,E2 -21300.06} C_VEL
LIN {X 0,Y 208.9,Z 419.361,A -85,B 0,C 180,E1 -21301.903,E2 -21301.903} C_VEL
LIN {X 0,Y 209.56,Z 432.892,A -85,B 0,C 180,E1 -21303.887,E2 -21303.887} C_VEL
LIN {X 0,Y 210.487,Z 447.003,A -85,B 0,C 180,E1 -21306.382,E2 -21306.382} C_VEL
LIN {X 0,Y 210.992,Z 453.702,A -85,B 0,C 180,E1 -21307.737,E2 -21307.737} C_VEL
LIN {X 0,Y 209.432,Z 464.847,A -85,B 0,C 180,E1 -21310.395,E2 -21310.395} C_VEL
LIN {X 0,Y 208.115,Z 474.91,A -85,B 0,C 180,E1 -21313.321,E2 -21313.321} C_VEL
LIN {X 0,Y 207.415,Z 482.803,A -85,B 0,C 180,E1 -21316.074,E2 -21316.074} C_VEL
LIN {X 0,Y 206.618,Z 486.08,A -85,B 0,C 180,E1 -21317.429,E2 -21317.429} C_VEL
LIN {X 0,Y 203.763,Z 490.55,A -85,B 0,C 180,E1 -21319.77,E2 -21319.77} C_VEL
LIN {X 0,Y 201.14,Z 494.485,A -85,B 0,C 180,E1 -21322.258,E2 -21322.258} C_VEL
LIN {X 0,Y 200.714,Z 496.837,A -85,B 0,C 180,E1 -21323.808,E2 -21323.808} C_VEL
LIN {X 0,Y 201.261,Z 501.176,A -85,B 0,C 180,E1 -21326.999,E2 -21326.999} C_VEL
LIN {X 0,Y 201.666,Z 504.186,A -85,B 0,C 180,E1 -21330.002,E2 -21330.002} C_VEL
LIN {X 0,Y 200.959,Z 505.374,A -85,B 0,C 180,E1 -21332.006,E2 -21332.006} C_VEL
LIN {X 0,Y 199.556,Z 506.624,A -85,B 0,C 180,E1 -21336.067,E2 -21336.067} C_VEL
LIN {X 0,Y 198.704,Z 506.606,A -85,B 0,C 180,E1 -21340.188,E2 -21340.188} C_VEL
LIN {X 0,Y 198.925,Z 505.527,A -85,B 0,C 180,E1 -21344.32,E2 -21344.32} C_VEL
LIN {X 0,Y 200.594,Z 503.094,A -85,B 0,C 180,E1 -21348.921,E2 -21348.921} C_VEL
LIN {X 0,Y 202.978,Z 500.373,A -85,B 0,C 180,E1 -21352.389,E2 -21352.389} C_VEL
LIN {X 0,Y 206.881,Z 496.324,A -85,B 0,C 180,E1 -21356.209,E2 -21356.209} C_VEL
LIN {X 0,Y 213.479,Z 489.966,A -85,B 0,C 180,E1 -21360.684,E2 -21360.684} C_VEL
LIN {X 0,Y 218.189,Z 485.449,A -85,B 0,C 180,E1 -21363.203,E2 -21363.203} C_VEL
LIN {X 0,Y 223.695,Z 480.319,A -85,B 0,C 180,E1 -21365.539,E2 -21365.539} C_VEL
LIN {X 0,Y 232.877,Z 470.791,A -85,B 0,C 180,E1 -21369.33,E2 -21369.33} C_VEL
LIN {X 0,Y 238.504,Z 464.586,A -85,B 0,C 180,E1 -21371.531,E2 -21371.531} C_VEL
LIN {X 0,Y 243.74,Z 458.273,A -85,B 0,C 180,E1 -21373.876,E2 -21373.876} C_VEL
LIN {X 0,Y 248.289,Z 452.59,A -85,B 0,C 180,E1 -21376.162,E2 -21376.162} C_VEL
LIN {X 0,Y 252.9,Z 447.115,A -85,B 0,C 180,E1 -21378.62,E2 -21378.62} C_VEL
LIN {X 0,Y 254.145,Z 445.153,A -85,B 0,C 180,E1 -21380.743,E2 -21380.743} C_VEL
LIN {X 0,Y 253.543,Z 445.234,A -85,B 0,C 180,E1 -21382.424,E2 -21382.424} C_VEL
LIN {X 0,Y 244.823,Z 451.304,A -85,B 0,C 180,E1 -21384.962,E2 -21384.962} C_VEL
LIN {X 0,Y 236.709,Z 456.166,A -85,B 0,C 180,E1 -21387.695,E2 -21387.695} C_VEL
LIN {X 0,Y 229.365,Z 459.858,A -85,B 0,C 180,E1 -21390.643,E2 -21390.643} C_VEL
LIN {X 0,Y 222.815,Z 462.436,A -85,B 0,C 180,E1 -21393.795,E2 -21393.795} C_VEL
LIN {X 0,Y 216.993,Z 463.958,A -85,B 0,C 180,E1 -21397.129,E2 -21397.129} C_VEL
LIN {X 0,Y 212.113,Z 464.384,A -85,B 0,C 180,E1 -21400.651,E2 -21400.651} C_VEL
LIN {X 0,Y 207.939,Z 463.77,A -85,B 0,C 180,E1 -21404.313,E2 -21404.313} C_VEL
LIN {X 0,Y 204.655,Z 462.024,A -85,B 0,C 180,E1 -21408.11,E2 -21408.11} C_VEL
LIN {X 0,Y 202.188,Z 459.125,A -85,B 0,C 180,E1 -21412.008,E2 -21412.008} C_VEL
LIN {X 0,Y 200.638,Z 455.021,A -85,B 0,C 180,E1 -21415.983,E2 -21415.983} C_VEL
LIN {X 0,Y 199.895,Z 449.64,A -85,B 0,C 180,E1 -21420.001,E2 -21420.001} C_VEL
LIN {X 0,Y 199.636,Z 444.689,A -85,B 0,C 180,E1 -21423.028,E2 -21423.028} C_VEL
LIN {X 0,Y 199.878,Z 436.672,A -85,B 0,C 180,E1 -21427.07,E2 -21427.07} C_VEL
LIN {X 0,Y 200.612,Z 429.501,A -85,B 0,C 180,E1 -21430.089,E2 -21430.089} C_VEL
LIN {X 0,Y 201.696,Z 419.576,A -85,B 0,C 180,E1 -21433.604,E2 -21433.604} C_VEL
LIN {X 0,Y 203.014,Z 409.508,A -85,B 0,C 180,E1 -21436.595,E2 -21436.595} C_VEL
LIN {X 0,Y 204.673,Z 397.625,A -85,B 0,C 180,E1 -21439.561,E2 -21439.561} C_VEL
LIN {X 0,Y 206.62,Z 384.749,A -85,B 0,C 180,E1 -21442.205,E2 -21442.205} C_VEL
LIN {X 0,Y 207.518,Z 378.187,A -85,B 0,C 180,E1 -21443.377,E2 -21443.377} C_VEL
LIN {X 0,Y 203.74,Z 363.717,A -85,B 0,C 180,E1 -21445.92,E2 -21445.92} C_VEL
LIN {X 0,Y 199.872,Z 348.82,A -85,B 0,C 180,E1 -21448.204,E2 -21448.204} C_VEL
LIN {X 0,Y 199.759,Z 348.268,A -85,B 0,C 180,E1 -21448.536,E2 -21448.536} C_VEL
LIN {X 0,Y 199.684,Z 348.238,A -85,B 0,C 180,E1 -21452.358,E2 -21452.358} C_VEL
LIN {X 0,Y 199.629,Z 348.241,A -85,B 0,C 180,E1 -21456.763,E2 -21456.763} C_VEL
LIN {X 0,Y 199.614,Z 348.243,A -85,B 0,C 180,E1 -21459.328,E2 -21459.328} C_VEL
LIN {X 0,Y 199.581,Z 348.25,A -85,B 0,C 180,E1 -21462.31,E2 -21462.31} C_VEL
LIN {X 0,Y 199.607,Z 348.241,A -85,B 0,C 180,E1 -21465.234,E2 -21465.234} C_VEL
LIN {X 0,Y 199.61,Z 348.245,A -85,B 0,C 180,E1 -21468.011,E2 -21468.011} C_VEL
LIN {X 0,Y 199.648,Z 348.24,A -85,B 0,C 180,E1 -21470.756,E2 -21470.756} C_VEL
LIN {X 0,Y 199.639,Z 348.239,A -85,B 0,C 180,E1 -21475.717,E2 -21475.717} C_VEL
LIN {X 0,Y 199.702,Z 348.236,A -85,B 0,C 180,E1 -21478.135,E2 -21478.135} C_VEL
LIN {X 0,Y 199.691,Z 348.232,A -85,B 0,C 180,E1 -21482.77,E2 -21482.77} C_VEL
LIN {X 0,Y 199.72,Z 348.23,A -85,B 0,C 180,E1 -21487.225,E2 -21487.225} C_VEL
LIN {X 0,Y 199.802,Z 348.218,A -85,B 0,C 180,E1 -21491.756,E2 -21491.756} C_VEL
LIN {X 0,Y 199.854,Z 348.216,A -85,B 0,C 180,E1 -21495.748,E2 -21495.748} C_VEL
LIN {X 0,Y 200.081,Z 348.184,A -85,B 0,C 180,E1 -21499.883,E2 -21499.883} C_VEL
LIN {X 0,Y 200.137,Z 348.181,A -85,B 0,C 180,E1 -21501.924,E2 -21501.924} C_VEL
LIN {X 0,Y 200.327,Z 348.154,A -85,B 0,C 180,E1 -21507.988,E2 -21507.988} C_VEL
LIN {X 0,Y 200.484,Z 348.137,A -85,B 0,C 180,E1 -21509.998,E2 -21509.998} C_VEL
LIN {X 0,Y 200.037,Z 348.191,A -85,B 0,C 180,E1 -21514.027,E2 -21514.027} C_VEL
LIN {X 0,Y 200.136,Z 348.179,A -85,B 0,C 180,E1 -21518.073,E2 -21518.073} C_VEL
LIN {X 0,Y 199.918,Z 348.205,A -85,B 0,C 180,E1 -21522.175,E2 -21522.175} C_VEL
LIN {X 0,Y 199.808,Z 348.218,A -85,B 0,C 180,E1 -21526.341,E2 -21526.341} C_VEL
LIN {X 0,Y 199.825,Z 348.217,A -85,B 0,C 180,E1 -21528.452,E2 -21528.452} C_VEL
LIN {X 0,Y 199.738,Z 348.226,A -85,B 0,C 180,E1 -21533.815,E2 -21533.815} C_VEL
LIN {X 0,Y 199.708,Z 348.232,A -85,B 0,C 180,E1 -21538.382,E2 -21538.382} C_VEL
LIN {X 0,Y 199.67,Z 348.232,A -85,B 0,C 180,E1 -21542.353,E2 -21542.353} C_VEL
LIN {X 0,Y 199.621,Z 348.244,A -85,B 0,C 180,E1 -21546.761,E2 -21546.761} C_VEL
LIN {X 0,Y 199.606,Z 348.243,A -85,B 0,C 180,E1 -21549.326,E2 -21549.326} C_VEL
LIN {X 0,Y 199.572,Z 348.247,A -85,B 0,C 180,E1 -21552.308,E2 -21552.308} C_VEL
LIN {X 0,Y 199.578,Z 348.25,A -85,B 0,C 180,E1 -21555.227,E2 -21555.227} C_VEL
LIN {X 0,Y 199.577,Z 348.246,A -85,B 0,C 180,E1 -21558.003,E2 -21558.003} C_VEL
LIN {X 0,Y 199.607,Z 348.244,A -85,B 0,C 180,E1 -21560.766,E2 -21560.766} C_VEL
LIN {X 0,Y 199.609,Z 348.243,A -85,B 0,C 180,E1 -21565.712,E2 -21565.712} C_VEL
LIN {X 0,Y 199.696,Z 348.229,A -85,B 0,C 180,E1 -21568.135,E2 -21568.135} C_VEL
LIN {X 0,Y 199.682,Z 348.238,A -85,B 0,C 180,E1 -21572.77,E2 -21572.77} C_VEL
LIN {X 0,Y 199.733,Z 348.228,A -85,B 0,C 180,E1 -21577.228,E2 -21577.228} C_VEL
LIN {X 0,Y 199.832,Z 348.216,A -85,B 0,C 180,E1 -21581.721,E2 -21581.721} C_VEL
LIN {X 0,Y 199.842,Z 348.212,A -85,B 0,C 180,E1 -21585.748,E2 -21585.748} C_VEL
LIN {X 0,Y 200.069,Z 348.187,A -85,B 0,C 180,E1 -21589.884,E2 -21589.884} C_VEL
LIN {X 0,Y 200.035,Z 348.188,A -85,B 0,C 180,E1 -21593.949,E2 -21593.949} C_VEL
LIN {X 0,Y 200.316,Z 348.157,A -85,B 0,C 180,E1 -21597.989,E2 -21597.989} C_VEL
LIN {X 0,Y 200.473,Z 348.137,A -85,B 0,C 180,E1 -21599.999,E2 -21599.999} C_VEL
LIN {X 0,Y 200.027,Z 348.192,A -85,B 0,C 180,E1 -21604.029,E2 -21604.029} C_VEL
LIN {X 0,Y 200.125,Z 348.182,A -85,B 0,C 180,E1 -21608.075,E2 -21608.075} C_VEL
LIN {X 0,Y 199.908,Z 348.207,A -85,B 0,C 180,E1 -21612.177,E2 -21612.177} C_VEL
LIN {X 0,Y 199.798,Z 348.222,A -85,B 0,C 180,E1 -21616.344,E2 -21616.344} C_VEL
LIN {X 0,Y 199.693,Z 348.233,A -85,B 0,C 180,E1 -21620.606,E2 -21620.606} C_VEL
LIN {X 0,Y 199.666,Z 348.236,A -85,B 0,C 180,E1 -21624.985,E2 -21624.985} C_VEL
LIN {X 0,Y 199.669,Z 348.236,A -85,B 0,C 180,E1 -21629.523,E2 -21629.523} C_VEL
LIN {X 0,Y 199.804,Z 348.333,A -85,B 0,C 180,E1 -21633.724,E2 -21633.724} C_VEL
LIN {X 0,Y 201.135,Z 355.359,A -85,B 0,C 180,E1 -21638.972,E2 -21638.972} C_VEL
LIN {X 0,Y 202.616,Z 362.339,A -85,B 0,C 180,E1 -21643.925,E2 -21643.925} C_VEL
LIN {X 0,Y 203.823,Z 368.082,A -85,B 0,C 180,E1 -21647.841,E2 -21647.841} C_VEL
LIN {X 0,Y 203.643,Z 370.425,A -85,B 0,C 180,E1 -21649.398,E2 -21649.398} C_VEL
LIN {X 0,Y 201.59,Z 378.783,A -85,B 0,C 180,E1 -21654.886,E2 -21654.886} C_VEL
LIN {X 0,Y 200.761,Z 383.514,A -85,B 0,C 180,E1 -21657.835,E2 -21657.835} C_VEL
LIN {X 0,Y 201.035,Z 401.468,A -85,B 0,C 180,E1 -21659.546,E2 -21659.546} C_VEL
LIN {X 0,Y 201.714,Z 417.736,A -85,B 0,C 180,E1 -21661.52,E2 -21661.52} C_VEL
LIN {X 0,Y 202.463,Z 432.326,A -85,B 0,C 180,E1 -21663.739,E2 -21663.739} C_VEL
LIN {X 0,Y 203.365,Z 446.306,A -85,B 0,C 180,E1 -21666.315,E2 -21666.315} C_VEL
LIN {X 0,Y 203.779,Z 454.164,A -85,B 0,C 180,E1 -21667.991,E2 -21667.991} C_VEL
LIN {X 0,Y 202.278,Z 464.911,A -85,B 0,C 180,E1 -21670.729,E2 -21670.729} C_VEL
LIN {X 0,Y 201.037,Z 474.739,A -85,B 0,C 180,E1 -21673.762,E2 -21673.762} C_VEL
LIN {X 0,Y 200.376,Z 482.975,A -85,B 0,C 180,E1 -21676.824,E2 -21676.824} C_VEL
LIN {X 0,Y 200.35,Z 490.88,A -85,B 0,C 180,E1 -21680.41,E2 -21680.41} C_VEL
LIN {X 0,Y 200.714,Z 496.837,A -85,B 0,C 180,E1 -21683.808,E2 -21683.808} C_VEL
LIN {X 0,Y 200.589,Z 498.337,A -85,B 0,C 180,E1 -21684.849,E2 -21684.849} C_VEL
LIN {X 0,Y 199.555,Z 500.122,A -85,B 0,C 180,E1 -21686.444,E2 -21686.444} C_VEL
LIN {X 0,Y 196.703,Z 502.123,A -85,B 0,C 180,E1 -21689.168,E2 -21689.168} C_VEL
LIN {X 0,Y 193.845,Z 503.708,A -85,B 0,C 180,E1 -21692.62,E2 -21692.62} C_VEL
LIN {X 0,Y 192.6,Z 504.904,A -85,B 0,C 180,E1 -21696.287,E2 -21696.287} C_VEL
LIN {X 0,Y 191.73,Z 505.103,A -85,B 0,C 180,E1 -21700.563,E2 -21700.563} C_VEL
LIN {X 0,Y 192.025,Z 504.269,A -85,B 0,C 180,E1 -21704.846,E2 -21704.846} C_VEL
LIN {X 0,Y 193.706,Z 502.233,A -85,B 0,C 180,E1 -21709.383,E2 -21709.383} C_VEL
LIN {X 0,Y 196.388,Z 499.608,A -85,B 0,C 180,E1 -21713.184,E2 -21713.184} C_VEL
LIN {X 0,Y 200.514,Z 495.919,A -85,B 0,C 180,E1 -21717.108,E2 -21717.108} C_VEL
LIN {X 0,Y 207.384,Z 489.993,A -85,B 0,C 180,E1 -21721.689,E2 -21721.689} C_VEL
LIN {X 0,Y 212.306,Z 485.733,A -85,B 0,C 180,E1 -21724.248,E2 -21724.248} C_VEL
LIN {X 0,Y 217.971,Z 480.973,A -85,B 0,C 180,E1 -21726.621,E2 -21726.621} C_VEL
LIN {X 0,Y 227.528,Z 472.05,A -85,B 0,C 180,E1 -21730.442,E2 -21730.442} C_VEL
LIN {X 0,Y 233.388,Z 466.251,A -85,B 0,C 180,E1 -21732.654,E2 -21732.654} C_VEL
LIN {X 0,Y 239.157,Z 460.017,A -85,B 0,C 180,E1 -21735.149,E2 -21735.149} C_VEL
LIN {X 0,Y 243.69,Z 454.965,A -85,B 0,C 180,E1 -21737.344,E2 -21737.344} C_VEL
LIN {X 0,Y 247.388,Z 451.05,A -85,B 0,C 180,E1 -21739.202,E2 -21739.202} C_VEL
LIN {X 0,Y 247.921,Z 450.284,A -85,B 0,C 180,E1 -21739.943,E2 -21739.943} C_VEL
LIN {X 0,Y 248.196,Z 449.5,A -85,B 0,C 180,E1 -21741.468,E2 -21741.468} C_VEL
LIN {X 0,Y 246.335,Z 450.632,A -85,B 0,C 180,E1 -21742.165,E2 -21742.165} C_VEL
LIN {X 0,Y 237.477,Z 455.9,A -85,B 0,C 180,E1 -21744.754,E2 -21744.754} C_VEL
LIN {X 0,Y 231.225,Z 459.133,A -85,B 0,C 180,E1 -21746.832,E2 -21746.832} C_VEL
LIN {X 0,Y 223.611,Z 462.423,A -85,B 0,C 180,E1 -21749.81,E2 -21749.81} C_VEL
LIN {X 0,Y 216.782,Z 464.639,A -85,B 0,C 180,E1 -21753.008,E2 -21753.008} C_VEL
LIN {X 0,Y 210.716,Z 465.821,A -85,B 0,C 180,E1 -21756.408,E2 -21756.408} C_VEL
LIN {X 0,Y 205.601,Z 465.931,A -85,B 0,C 180,E1 -21760.012,E2 -21760.012} C_VEL
LIN {X 0,Y 201.236,Z 464.998,A -85,B 0,C 180,E1 -21763.776,E2 -21763.776} C_VEL
LIN {X 0,Y 197.798,Z 462.945,A -85,B 0,C 180,E1 -21767.691,E2 -21767.691} C_VEL
LIN {X 0,Y 195.188,Z 459.76,A -85,B 0,C 180,E1 -21771.72,E2 -21771.72} C_VEL
LIN {X 0,Y 193.566,Z 455.379,A -85,B 0,C 180,E1 -21775.836,E2 -21775.836} C_VEL
LIN {X 0,Y 192.806,Z 449.721,A -85,B 0,C 180,E1 -21780.001,E2 -21780.001} C_VEL
LIN {X 0,Y 192.527,Z 444.509,A -85,B 0,C 180,E1 -21783.139,E2 -21783.139} C_VEL
LIN {X 0,Y 192.826,Z 436.211,A -85,B 0,C 180,E1 -21787.33,E2 -21787.33} C_VEL
LIN {X 0,Y 193.569,Z 428.756,A -85,B 0,C 180,E1 -21790.46,E2 -21790.46} C_VEL
LIN {X 0,Y 194.744,Z 418.503,A -85,B 0,C 180,E1 -21794.1,E2 -21794.1} C_VEL
LIN {X 0,Y 196.157,Z 408.064,A -85,B 0,C 180,E1 -21797.193,E2 -21797.193} C_VEL
LIN {X 0,Y 197.948,Z 395.674,A -85,B 0,C 180,E1 -21800.254,E2 -21800.254} C_VEL
LIN {X 0,Y 200.097,Z 381.899,A -85,B 0,C 180,E1 -21803.064,E2 -21803.064} C_VEL
LIN {X 0,Y 200.346,Z 378.791,A -85,B 0,C 180,E1 -21803.625,E2 -21803.625} C_VEL
LIN {X 0,Y 196.731,Z 364.783,A -85,B 0,C 180,E1 -21806.162,E2 -21806.162} C_VEL
LIN {X 0,Y 192.807,Z 349.584,A -85,B 0,C 180,E1 -21808.595,E2 -21808.595} C_VEL
LIN {X 0,Y 192.695,Z 349.146,A -85,B 0,C 180,E1 -21808.912,E2 -21808.912} C_VEL
LIN {X 0,Y 192.605,Z 349.118,A -85,B 0,C 180,E1 -21813.185,E2 -21813.185} C_VEL
LIN {X 0,Y 192.557,Z 349.122,A -85,B 0,C 180,E1 -21818.351,E2 -21818.351} C_VEL
LIN {X 0,Y 192.522,Z 349.126,A -85,B 0,C 180,E1 -21823.103,E2 -21823.103} C_VEL
LIN {X 0,Y 192.539,Z 349.125,A -85,B 0,C 180,E1 -21826.89,E2 -21826.89} C_VEL
LIN {X 0,Y 192.581,Z 349.119,A -85,B 0,C 180,E1 -21831.653,E2 -21831.653} C_VEL
LIN {X 0,Y 192.604,Z 349.115,A -85,B 0,C 180,E1 -21834.278,E2 -21834.278} C_VEL
LIN {X 0,Y 192.606,Z 349.116,A -85,B 0,C 180,E1 -21839.278,E2 -21839.278} C_VEL
LIN {X 0,Y 192.666,Z 349.107,A -85,B 0,C 180,E1 -21841.69,E2 -21841.69} C_VEL
LIN {X 0,Y 192.691,Z 349.108,A -85,B 0,C 180,E1 -21846.345,E2 -21846.345} C_VEL
LIN {X 0,Y 192.737,Z 349.097,A -85,B 0,C 180,E1 -21851.456,E2 -21851.456} C_VEL
LIN {X 0,Y 192.778,Z 349.095,A -85,B 0,C 180,E1 -21855.213,E2 -21855.213} C_VEL
LIN {X 0,Y 193.025,Z 349.062,A -85,B 0,C 180,E1 -21859.509,E2 -21859.509} C_VEL
LIN {X 0,Y 193.009,Z 349.069,A -85,B 0,C 180,E1 -21863.727,E2 -21863.727} C_VEL
LIN {X 0,Y 193.269,Z 349.032,A -85,B 0,C 180,E1 -21867.914,E2 -21867.914} C_VEL
LIN {X 0,Y 193.448,Z 349.013,A -85,B 0,C 180,E1 -21869.998,E2 -21869.998} C_VEL
LIN {X 0,Y 192.984,Z 349.069,A -85,B 0,C 180,E1 -21874.175,E2 -21874.175} C_VEL
LIN {X 0,Y 193.083,Z 349.056,A -85,B 0,C 180,E1 -21878.37,E2 -21878.37} C_VEL
LIN {X 0,Y 192.856,Z 349.085,A -85,B 0,C 180,E1 -21882.628,E2 -21882.628} C_VEL
LIN {X 0,Y 192.783,Z 349.095,A -85,B 0,C 180,E1 -21888.584,E2 -21888.584} C_VEL
LIN {X 0,Y 192.665,Z 349.106,A -85,B 0,C 180,E1 -21894.222,E2 -21894.222} C_VEL
LIN {X 0,Y 192.644,Z 349.113,A -85,B 0,C 180,E1 -21898.887,E2 -21898.887} C_VEL
LIN {X 0,Y 192.595,Z 349.117,A -85,B 0,C 180,E1 -21903.184,E2 -21903.184} C_VEL
LIN {X 0,Y 192.549,Z 349.123,A -85,B 0,C 180,E1 -21908.35,E2 -21908.35} C_VEL
LIN {X 0,Y 192.51,Z 349.13,A -85,B 0,C 180,E1 -21913.101,E2 -21913.101} C_VEL
LIN {X 0,Y 192.51,Z 349.131,A -85,B 0,C 180,E1 -21916.895,E2 -21916.895} C_VEL
LIN {X 0,Y 192.547,Z 349.124,A -85,B 0,C 180,E1 -21921.646,E2 -21921.646} C_VEL
LIN {X 0,Y 192.594,Z 349.117,A -85,B 0,C 180,E1 -21926.813,E2 -21926.813} C_VEL
LIN {X 0,Y 192.66,Z 349.11,A -85,B 0,C 180,E1 -21931.69,E2 -21931.69} C_VEL
LIN {X 0,Y 192.701,Z 349.102,A -85,B 0,C 180,E1 -21936.347,E2 -21936.347} C_VEL
LIN {X 0,Y 192.776,Z 349.095,A -85,B 0,C 180,E1 -21941.413,E2 -21941.413} C_VEL
LIN {X 0,Y 192.847,Z 349.086,A -85,B 0,C 180,E1 -21947.369,E2 -21947.369} C_VEL
LIN {X 0,Y 193.073,Z 349.057,A -85,B 0,C 180,E1 -21951.627,E2 -21951.627} C_VEL
LIN {X 0,Y 193.258,Z 349.036,A -85,B 0,C 180,E1 -21957.915,E2 -21957.915} C_VEL
LIN {X 0,Y 193.437,Z 349.014,A -85,B 0,C 180,E1 -21959.999,E2 -21959.999} C_VEL
LIN {X 0,Y 192.974,Z 349.071,A -85,B 0,C 180,E1 -21964.177,E2 -21964.177} C_VEL
LIN {X 0,Y 193.072,Z 349.059,A -85,B 0,C 180,E1 -21968.372,E2 -21968.372} C_VEL
LIN {X 0,Y 192.847,Z 349.087,A -85,B 0,C 180,E1 -21972.63,E2 -21972.63} C_VEL
LIN {X 0,Y 192.751,Z 349.097,A -85,B 0,C 180,E1 -21976.959,E2 -21976.959} C_VEL
LIN {X 0,Y 192.63,Z 349.113,A -85,B 0,C 180,E1 -21981.398,E2 -21981.398} C_VEL
LIN {X 0,Y 192.658,Z 349.112,A -85,B 0,C 180,E1 -21984.225,E2 -21984.225} C_VEL
LIN {X 0,Y 192.644,Z 349.11,A -85,B 0,C 180,E1 -21988.893,E2 -21988.893} C_VEL
LIN {X 0,Y 192.768,Z 349.189,A -85,B 0,C 180,E1 -21993.621,E2 -21993.621} C_VEL
LIN {X 0,Y 193.826,Z 354.895,A -85,B 0,C 180,E1 -21998.054,E2 -21998.054} C_VEL
LIN {X 0,Y 195.271,Z 361.765,A -85,B 0,C 180,E1 -22003.143,E2 -22003.143} C_VEL
LIN {X 0,Y 196.639,Z 367.514,A -85,B 0,C 180,E1 -22007.232,E2 -22007.232} C_VEL
LIN {X 0,Y 196.686,Z 369.523,A -85,B 0,C 180,E1 -22008.622,E2 -22008.622} C_VEL
LIN {X 0,Y 195.393,Z 374.917,A -85,B 0,C 180,E1 -22012.307,E2 -22012.307} C_VEL
LIN {X 0,Y 193.761,Z 382.505,A -85,B 0,C 180,E1 -22017.389,E2 -22017.389} C_VEL
LIN {X 0,Y 193.961,Z 400.94,A -85,B 0,C 180,E1 -22019.218,E2 -22019.218} C_VEL
LIN {X 0,Y 194.595,Z 416.485,A -85,B 0,C 180,E1 -22021.186,E2 -22021.186} C_VEL
LIN {X 0,Y 195.325,Z 431.243,A -85,B 0,C 180,E1 -22023.515,E2 -22023.515} C_VEL
LIN {X 0,Y 196.21,Z 445.447,A -85,B 0,C 180,E1 -22026.239,E2 -22026.239} C_VEL
LIN {X 0,Y 196.692,Z 453.685,A -85,B 0,C 180,E1 -22028.077,E2 -22028.077} C_VEL
LIN {X 0,Y 195.108,Z 464.854,A -85,B 0,C 180,E1 -22031.086,E2 -22031.086} C_VEL
LIN {X 0,Y 193.996,Z 474.485,A -85,B 0,C 180,E1 -22034.236,E2 -22034.236} C_VEL
LIN {X 0,Y 193.406,Z 482.525,A -85,B 0,C 180,E1 -22037.409,E2 -22037.409} C_VEL
LIN {X 0,Y 193.464,Z 489.246,A -85,B 0,C 180,E1 -22040.593,E2 -22040.593} C_VEL
LIN {X 0,Y 193.879,Z 495.218,A -85,B 0,C 180,E1 -22044.091,E2 -22044.091} C_VEL
LIN {X 0,Y 194.364,Z 499.052,A -85,B 0,C 180,E1 -22046.893,E2 -22046.893} C_VEL
LIN {X 0,Y 194.804,Z 502.197,A -85,B 0,C 180,E1 -22050.002,E2 -22050.002} C_VEL
LIN {X 0,Y 193.845,Z 503.708,A -85,B 0,C 180,E1 -22052.62,E2 -22052.62} C_VEL
LIN {X 0,Y 192.523,Z 504.219,A -85,B 0,C 180,E1 -22054.32,E2 -22054.32} C_VEL
LIN {X 0,Y 188.844,Z 504.162,A -85,B 0,C 180,E1 -22057.09,E2 -22057.09} C_VEL
LIN {X 0,Y 186.02,Z 503.786,A -85,B 0,C 180,E1 -22059.375,E2 -22059.375} C_VEL
LIN {X 0,Y 184.846,Z 503.532,A -85,B 0,C 180,E1 -22061.177,E2 -22061.177} C_VEL
LIN {X 0,Y 184.754,Z 503.442,A -85,B 0,C 180,E1 -22061.791,E2 -22061.791} C_VEL
LIN {X 0,Y 185.148,Z 502.881,A -85,B 0,C 180,E1 -22065.411,E2 -22065.411} C_VEL
LIN {X 0,Y 186.86,Z 501.256,A -85,B 0,C 180,E1 -22069.903,E2 -22069.903} C_VEL
LIN {X 0,Y 189.819,Z 498.787,A -85,B 0,C 180,E1 -22074.036,E2 -22074.036} C_VEL
LIN {X 0,Y 195.496,Z 494.412,A -85,B 0,C 180,E1 -22079.035,E2 -22079.035} C_VEL
LIN {X 0,Y 202.964,Z 488.669,A -85,B 0,C 180,E1 -22083.646,E2 -22083.646} C_VEL
LIN {X 0,Y 212.344,Z 481.556,A -85,B 0,C 180,E1 -22087.758,E2 -22087.758} C_VEL
LIN {X 0,Y 222.245,Z 473.222,A -85,B 0,C 180,E1 -22091.613,E2 -22091.613} C_VEL
LIN {X 0,Y 228.322,Z 467.788,A -85,B 0,C 180,E1 -22093.836,E2 -22093.836} C_VEL
LIN {X 0,Y 234.568,Z 461.733,A -85,B 0,C 180,E1 -22096.44,E2 -22096.44} C_VEL
LIN {X 0,Y 240.785,Z 455.64,A -85,B 0,C 180,E1 -22099.368,E2 -22099.368} C_VEL
LIN {X 0,Y 242.167,Z 454.214,A -85,B 0,C 180,E1 -22100.323,E2 -22100.323} C_VEL
LIN {X 0,Y 241.407,Z 454.32,A -85,B 0,C 180,E1 -22101.25,E2 -22101.25} C_VEL
LIN {X 0,Y 232.246,Z 459.114,A -85,B 0,C 180,E1 -22103.837,E2 -22103.837} C_VEL
LIN {X 0,Y 225.775,Z 462.016,A -85,B 0,C 180,E1 -22105.923,E2 -22105.923} C_VEL
LIN {X 0,Y 217.879,Z 464.899,A -85,B 0,C 180,E1 -22108.929,E2 -22108.929} C_VEL
LIN {X 0,Y 210.757,Z 466.738,A -85,B 0,C 180,E1 -22112.17,E2 -22112.17} C_VEL
LIN {X 0,Y 204.429,Z 467.568,A -85,B 0,C 180,E1 -22115.636,E2 -22115.636} C_VEL
LIN {X 0,Y 199.082,Z 467.351,A -85,B 0,C 180,E1 -22119.328,E2 -22119.328} C_VEL
LIN {X 0,Y 194.513,Z 466.105,A -85,B 0,C 180,E1 -22123.199,E2 -22123.199} C_VEL
LIN {X 0,Y 190.927,Z 463.75,A -85,B 0,C 180,E1 -22127.241,E2 -22127.241} C_VEL
LIN {X 0,Y 188.183,Z 460.273,A -85,B 0,C 180,E1 -22131.409,E2 -22131.409} C_VEL
LIN {X 0,Y 186.49,Z 455.597,A -85,B 0,C 180,E1 -22135.678,E2 -22135.678} C_VEL
LIN {X 0,Y 185.719,Z 449.634,A -85,B 0,C 180,E1 -22140.001,E2 -22140.001} C_VEL
LIN {X 0,Y 185.401,Z 442.217,A -85,B 0,C 180,E1 -22144.349,E2 -22144.349} C_VEL
LIN {X 0,Y 186.07,Z 433.171,A -85,B 0,C 180,E1 -22148.69,E2 -22148.69} C_VEL
LIN {X 0,Y 187.107,Z 423.26,A -85,B 0,C 180,E1 -22152.573,E2 -22152.573} C_VEL
LIN {X 0,Y 188.56,Z 412.029,A -85,B 0,C 180,E1 -22156.233,E2 -22156.233} C_VEL
LIN {X 0,Y 190.363,Z 399.205,A -85,B 0,C 180,E1 -22159.688,E2 -22159.688} C_VEL
LIN {X 0,Y 192.36,Z 386.176,A -85,B 0,C 180,E1 -22162.559,E2 -22162.559} C_VEL
LIN {X 0,Y 193.318,Z 380.217,A -85,B 0,C 180,E1 -22163.696,E2 -22163.696} C_VEL
LIN {X 0,Y 189.68,Z 365.857,A -85,B 0,C 180,E1 -22166.4,E2 -22166.4} C_VEL
LIN {X 0,Y 185.768,Z 350.584,A -85,B 0,C 180,E1 -22168.899,E2 -22168.899} C_VEL
LIN {X 0,Y 185.624,Z 350.04,A -85,B 0,C 180,E1 -22169.236,E2 -22169.236} C_VEL
LIN {X 0,Y 185.506,Z 350.003,A -85,B 0,C 180,E1 -22174.632,E2 -22174.632} C_VEL
LIN {X 0,Y 185.511,Z 349.998,A -85,B 0,C 180,E1 -22177.313,E2 -22177.313} C_VEL
LIN {X 0,Y 185.477,Z 350.007,A -85,B 0,C 180,E1 -22180.724,E2 -22180.724} C_VEL
LIN {X 0,Y 185.504,Z 349.998,A -85,B 0,C 180,E1 -22186.042,E2 -22186.042} C_VEL
LIN {X 0,Y 185.503,Z 350.002,A -85,B 0,C 180,E1 -22189.902,E2 -22189.902} C_VEL
LIN {X 0,Y 185.55,Z 349.993,A -85,B 0,C 180,E1 -22192.695,E2 -22192.695} C_VEL
LIN {X 0,Y 185.547,Z 349.998,A -85,B 0,C 180,E1 -22197.974,E2 -22197.974} C_VEL
LIN {X 0,Y 185.586,Z 349.989,A -85,B 0,C 180,E1 -22200.576,E2 -22200.576} C_VEL
LIN {X 0,Y 185.585,Z 349.991,A -85,B 0,C 180,E1 -22205.38,E2 -22205.38} C_VEL
LIN {X 0,Y 185.68,Z 349.975,A -85,B 0,C 180,E1 -22211.132,E2 -22211.132} C_VEL
LIN {X 0,Y 185.73,Z 349.974,A -85,B 0,C 180,E1 -22214.638,E2 -22214.638} C_VEL
LIN {X 0,Y 185.948,Z 349.942,A -85,B 0,C 180,E1 -22219.327,E2 -22219.327} C_VEL
LIN {X 0,Y 185.974,Z 349.944,A -85,B 0,C 180,E1 -22223.488,E2 -22223.488} C_VEL
LIN {X 0,Y 186.213,Z 349.911,A -85,B 0,C 180,E1 -22227.835,E2 -22227.835} C_VEL
LIN {X 0,Y 186.411,Z 349.89,A -85,B 0,C 180,E1 -22229.998,E2 -22229.998} C_VEL
LIN {X 0,Y 185.931,Z 349.947,A -85,B 0,C 180,E1 -22234.334,E2 -22234.334} C_VEL
LIN {X 0,Y 186.033,Z 349.934,A -85,B 0,C 180,E1 -22238.689,E2 -22238.689} C_VEL
LIN {X 0,Y 185.768,Z 349.969,A -85,B 0,C 180,E1 -22243.118,E2 -22243.118} C_VEL
LIN {X 0,Y 185.719,Z 349.977,A -85,B 0,C 180,E1 -22247.62,E2 -22247.62} C_VEL
LIN {X 0,Y 185.601,Z 349.987,A -85,B 0,C 180,E1 -22252.248,E2 -22252.248} C_VEL
LIN {X 0,Y 185.561,Z 349.995,A -85,B 0,C 180,E1 -22257.03,E2 -22257.03} C_VEL
LIN {X 0,Y 185.577,Z 349.993,A -85,B 0,C 180,E1 -22259.491,E2 -22259.491} C_VEL
LIN {X 0,Y 185.497,Z 350.002,A -85,B 0,C 180,E1 -22264.63,E2 -22264.63} C_VEL
LIN {X 0,Y 185.504,Z 350.003,A -85,B 0,C 180,E1 -22267.311,E2 -22267.311} C_VEL
LIN {X 0,Y 185.469,Z 350.003,A -85,B 0,C 180,E1 -22270.723,E2 -22270.723} C_VEL
LIN {X 0,Y 185.46,Z 350.007,A -85,B 0,C 180,E1 -22273.944,E2 -22273.944} C_VEL
LIN {X 0,Y 185.473,Z 350.006,A -85,B 0,C 180,E1 -22276.994,E2 -22276.994} C_VEL
LIN {X 0,Y 185.465,Z 350.003,A -85,B 0,C 180,E1 -22279.893,E2 -22279.893} C_VEL
LIN {X 0,Y 185.502,Z 350.003,A -85,B 0,C 180,E1 -22282.709,E2 -22282.709} C_VEL
LIN {X 0,Y 185.542,Z 349.992,A -85,B 0,C 180,E1 -22287.974,E2 -22287.974} C_VEL
LIN {X 0,Y 185.577,Z 349.993,A -85,B 0,C 180,E1 -22290.574,E2 -22290.574} C_VEL
LIN {X 0,Y 185.583,Z 349.988,A -85,B 0,C 180,E1 -22295.381,E2 -22295.381} C_VEL
LIN {X 0,Y 185.688,Z 349.979,A -85,B 0,C 180,E1 -22301.114,E2 -22301.114} C_VEL
LIN {X 0,Y 185.722,Z 349.972,A -85,B 0,C 180,E1 -22304.639,E2 -22304.639} C_VEL
LIN {X 0,Y 185.937,Z 349.948,A -85,B 0,C 180,E1 -22309.327,E2 -22309.327} C_VEL
LIN {X 0,Y 185.963,Z 349.939,A -85,B 0,C 180,E1 -22313.489,E2 -22313.489} C_VEL
LIN {X 0,Y 186.203,Z 349.915,A -85,B 0,C 180,E1 -22317.836,E2 -22317.836} C_VEL
LIN {X 0,Y 186.4,Z 349.89,A -85,B 0,C 180,E1 -22319.999,E2 -22319.999} C_VEL
LIN {X 0,Y 185.922,Z 349.951,A -85,B 0,C 180,E1 -22324.335,E2 -22324.335} C_VEL
LIN {X 0,Y 186.022,Z 349.935,A -85,B 0,C 180,E1 -22328.691,E2 -22328.691} C_VEL
LIN {X 0,Y 185.758,Z 349.969,A -85,B 0,C 180,E1 -22333.12,E2 -22333.12} C_VEL
LIN {X 0,Y 185.683,Z 349.978,A -85,B 0,C 180,E1 -22337.625,E2 -22337.625} C_VEL
LIN {X 0,Y 185.59,Z 349.993,A -85,B 0,C 180,E1 -22342.252,E2 -22342.252} C_VEL
LIN {X 0,Y 185.556,Z 349.991,A -85,B 0,C 180,E1 -22347.033,E2 -22347.033} C_VEL
LIN {X 0,Y 185.596,Z 349.992,A -85,B 0,C 180,E1 -22352.014,E2 -22352.014} C_VEL
LIN {X 0,Y 185.737,Z 350.128,A -85,B 0,C 180,E1 -22353.653,E2 -22353.653} C_VEL
LIN {X 0,Y 186.911,Z 356.334,A -85,B 0,C 180,E1 -22358.612,E2 -22358.612} C_VEL
LIN {X 0,Y 188.349,Z 362.916,A -85,B 0,C 180,E1 -22363.639,E2 -22363.639} C_VEL
LIN {X 0,Y 189.624,Z 368.631,A -85,B 0,C 180,E1 -22367.838,E2 -22367.838} C_VEL
LIN {X 0,Y 188.84,Z 372.727,A -85,B 0,C 180,E1 -22370.755,E2 -22370.755} C_VEL
LIN {X 0,Y 186.79,Z 381.342,A -85,B 0,C 180,E1 -22376.859,E2 -22376.859} C_VEL
LIN {X 0,Y 186.743,Z 382.633,A -85,B 0,C 180,E1 -22377.091,E2 -22377.091} C_VEL
LIN {X 0,Y 186.838,Z 398.642,A -85,B 0,C 180,E1 -22378.692,E2 -22378.692} C_VEL
LIN {X 0,Y 187.438,Z 415.001,A -85,B 0,C 180,E1 -22380.83,E2 -22380.83} C_VEL
LIN {X 0,Y 188.084,Z 428.802,A -85,B 0,C 180,E1 -22383.062,E2 -22383.062} C_VEL
LIN {X 0,Y 188.949,Z 442.998,A -85,B 0,C 180,E1 -22385.851,E2 -22385.851} C_VEL
LIN {X 0,Y 189.671,Z 451.885,A -85,B 0,C 180,E1 -22387.871,E2 -22387.871} C_VEL
LIN {X 0,Y 188.219,Z 462.965,A -85,B 0,C 180,E1 -22390.932,E2 -22390.932} C_VEL
LIN {X 0,Y 187.092,Z 472.658,A -85,B 0,C 180,E1 -22394.199,E2 -22394.199} C_VEL
LIN {X 0,Y 186.502,Z 482.004,A -85,B 0,C 180,E1 -22398.042,E2 -22398.042} C_VEL
LIN {X 0,Y 186.648,Z 488.567,A -85,B 0,C 180,E1 -22401.339,E2 -22401.339} C_VEL
LIN {X 0,Y 187.113,Z 493.875,A -85,B 0,C 180,E1 -22404.614,E2 -22404.614} C_VEL
LIN {X 0,Y 187.674,Z 498.044,A -85,B 0,C 180,E1 -22407.856,E2 -22407.856} C_VEL
LIN {X 0,Y 187.956,Z 500.159,A -85,B 0,C 180,E1 -22410.002,E2 -22410.002} C_VEL
LIN {X 0,Y 187.071,Z 501.669,A -85,B 0,C 180,E1 -22412.439,E2 -22412.439} C_VEL
LIN {X 0,Y 185.634,Z 503.155,A -85,B 0,C 180,E1 -22416.524,E2 -22416.524} C_VEL
LIN {X 0,Y 184.774,Z 503.515,A -85,B 0,C 180,E1 -22420.965,E2 -22420.965} C_VEL
LIN {X 0,Y 184.754,Z 503.442,A -85,B 0,C 180,E1 -22421.791,E2 -22421.791} C_VEL
LIN {X 0,Y 184.193,Z 503.128,A -85,B 0,C 180,E1 -22423.616,E2 -22423.616} C_VEL
LIN {X 0,Y 181.946,Z 501.989,A -85,B 0,C 180,E1 -22426.622,E2 -22426.622} C_VEL
LIN {X 0,Y 180.304,Z 500.537,A -85,B 0,C 180,E1 -22429.681,E2 -22429.681} C_VEL
LIN {X 0,Y 180.697,Z 499.664,A -85,B 0,C 180,E1 -22431.531,E2 -22431.531} C_VEL
LIN {X 0,Y 185.406,Z 496.461,A -85,B 0,C 180,E1 -22437.059,E2 -22437.059} C_VEL
LIN {X 0,Y 192.212,Z 491.958,A -85,B 0,C 180,E1 -22442.019,E2 -22442.019} C_VEL
LIN {X 0,Y 200.753,Z 486.144,A -85,B 0,C 180,E1 -22446.524,E2 -22446.524} C_VEL
LIN {X 0,Y 206.787,Z 482,A -85,B 0,C 180,E1 -22448.96,E2 -22448.96} C_VEL
LIN {X 0,Y 217.061,Z 474.243,A -85,B 0,C 180,E1 -22452.841,E2 -22452.841} C_VEL
LIN {X 0,Y 223.337,Z 469.18,A -85,B 0,C 180,E1 -22455.077,E2 -22455.077} C_VEL
LIN {X 0,Y 229.913,Z 463.459,A -85,B 0,C 180,E1 -22457.74,E2 -22457.74} C_VEL
LIN {X 0,Y 234.279,Z 459.602,A -85,B 0,C 180,E1 -22459.71,E2 -22459.71} C_VEL
LIN {X 0,Y 235.447,Z 458.447,A -85,B 0,C 180,E1 -22460.569,E2 -22460.569} C_VEL
LIN {X 0,Y 224.806,Z 463.163,A -85,B 0,C 180,E1 -22463.56,E2 -22463.56} C_VEL
LIN {X 0,Y 216.163,Z 466.197,A -85,B 0,C 180,E1 -22466.447,E2 -22466.447} C_VEL
LIN {X 0,Y 208.405,Z 468.167,A -85,B 0,C 180,E1 -22469.613,E2 -22469.613} C_VEL
LIN {X 0,Y 201.356,Z 469.171,A -85,B 0,C 180,E1 -22473.016,E2 -22473.016} C_VEL
LIN {X 0,Y 195.308,Z 469.134,A -85,B 0,C 180,E1 -22476.683,E2 -22476.683} C_VEL
LIN {X 0,Y 190.111,Z 468.081,A -85,B 0,C 180,E1 -22480.567,E2 -22480.567} C_VEL
LIN {X 0,Y 185.868,Z 465.953,A -85,B 0,C 180,E1 -22484.652,E2 -22484.652} C_VEL
LIN {X 0,Y 182.487,Z 462.743,A -85,B 0,C 180,E1 -22488.898,E2 -22488.898} C_VEL
LIN {X 0,Y 180.173,Z 458.378,A -85,B 0,C 180,E1 -22493.28,E2 -22493.28} C_VEL
LIN {X 0,Y 178.878,Z 452.785,A -85,B 0,C 180,E1 -22497.749,E2 -22497.749} C_VEL
LIN {X 0,Y 178.561,Z 447.681,A -85,B 0,C 180,E1 -22501.128,E2 -22501.128} C_VEL
LIN {X 0,Y 178.322,Z 439.531,A -85,B 0,C 180,E1 -22505.655,E2 -22505.655} C_VEL
LIN {X 0,Y 179.218,Z 430.987,A -85,B 0,C 180,E1 -22509.594,E2 -22509.594} C_VEL
LIN {X 0,Y 180.29,Z 420.791,A -85,B 0,C 180,E1 -22513.527,E2 -22513.527} C_VEL
LIN {X 0,Y 181.963,Z 408.49,A -85,B 0,C 180,E1 -22517.418,E2 -22517.418} C_VEL
LIN {X 0,Y 183.81,Z 395.93,A -85,B 0,C 180,E1 -22520.713,E2 -22520.713} C_VEL
LIN {X 0,Y 186.021,Z 382.109,A -85,B 0,C 180,E1 -22523.668,E2 -22523.668} C_VEL
LIN {X 0,Y 186.163,Z 380.671,A -85,B 0,C 180,E1 -22523.944,E2 -22523.944} C_VEL
LIN {X 0,Y 182.667,Z 367.014,A -85,B 0,C 180,E1 -22526.602,E2 -22526.602} C_VEL
LIN {X 0,Y 178.664,Z 351.432,A -85,B 0,C 180,E1 -22529.268,E2 -22529.268} C_VEL
LIN {X 0,Y 178.549,Z 350.886,A -85,B 0,C 180,E1 -22529.787,E2 -22529.787} C_VEL
LIN {X 0,Y 178.491,Z 350.877,A -85,B 0,C 180,E1 -22534.219,E2 -22534.219} C_VEL
LIN {X 0,Y 178.402,Z 350.886,A -85,B 0,C 180,E1 -22539.074,E2 -22539.074} C_VEL
LIN {X 0,Y 178.414,Z 350.886,A -85,B 0,C 180,E1 -22542.041,E2 -22542.041} C_VEL
LIN {X 0,Y 178.425,Z 350.879,A -85,B 0,C 180,E1 -22545.155,E2 -22545.155} C_VEL
LIN {X 0,Y 178.43,Z 350.885,A -85,B 0,C 180,E1 -22548.451,E2 -22548.451} C_VEL
LIN {X 0,Y 178.455,Z 350.876,A -85,B 0,C 180,E1 -22553.789,E2 -22553.789} C_VEL
LIN {X 0,Y 178.495,Z 350.876,A -85,B 0,C 180,E1 -22556.546,E2 -22556.546} C_VEL
LIN {X 0,Y 178.527,Z 350.872,A -85,B 0,C 180,E1 -22560.006,E2 -22560.006} C_VEL
LIN {X 0,Y 178.525,Z 350.87,A -85,B 0,C 180,E1 -22564.885,E2 -22564.885} C_VEL
LIN {X 0,Y 178.628,Z 350.853,A -85,B 0,C 180,E1 -22570.783,E2 -22570.783} C_VEL
LIN {X 0,Y 178.671,Z 350.855,A -85,B 0,C 180,E1 -22574.015,E2 -22574.015} C_VEL
LIN {X 0,Y 178.9,Z 350.82,A -85,B 0,C 180,E1 -22579.151,E2 -22579.151} C_VEL
LIN {X 0,Y 178.939,Z 350.82,A -85,B 0,C 180,E1 -22583.231,E2 -22583.231} C_VEL
LIN {X 0,Y 179.159,Z 350.789,A -85,B 0,C 180,E1 -22587.75,E2 -22587.75} C_VEL
LIN {X 0,Y 179.374,Z 350.766,A -85,B 0,C 180,E1 -22589.998,E2 -22589.998} C_VEL
LIN {X 0,Y 178.88,Z 350.825,A -85,B 0,C 180,E1 -22594.505,E2 -22594.505} C_VEL
LIN {X 0,Y 178.982,Z 350.813,A -85,B 0,C 180,E1 -22599.035,E2 -22599.035} C_VEL
LIN {X 0,Y 178.691,Z 350.848,A -85,B 0,C 180,E1 -22603.647,E2 -22603.647} C_VEL
LIN {X 0,Y 178.672,Z 350.852,A -85,B 0,C 180,E1 -22608.339,E2 -22608.339} C_VEL
LIN {X 0,Y 178.514,Z 350.87,A -85,B 0,C 180,E1 -22613.182,E2 -22613.182} C_VEL
LIN {X 0,Y 178.486,Z 350.876,A -85,B 0,C 180,E1 -22618.195,E2 -22618.195} C_VEL
LIN {X 0,Y 178.476,Z 350.876,A -85,B 0,C 180,E1 -22620.789,E2 -22620.789} C_VEL
LIN {X 0,Y 178.483,Z 350.875,A -85,B 0,C 180,E1 -22624.217,E2 -22624.217} C_VEL
LIN {X 0,Y 178.394,Z 350.887,A -85,B 0,C 180,E1 -22629.072,E2 -22629.072} C_VEL
LIN {X 0,Y 178.405,Z 350.884,A -85,B 0,C 180,E1 -22632.04,E2 -22632.04} C_VEL
LIN {X 0,Y 178.393,Z 350.889,A -85,B 0,C 180,E1 -22635.161,E2 -22635.161} C_VEL
LIN {X 0,Y 178.404,Z 350.884,A -85,B 0,C 180,E1 -22638.455,E2 -22638.455} C_VEL
LIN {X 0,Y 178.419,Z 350.884,A -85,B 0,C 180,E1 -22643.781,E2 -22643.781} C_VEL
LIN {X 0,Y 178.483,Z 350.876,A -85,B 0,C 180,E1 -22646.545,E2 -22646.545} C_VEL
LIN {X 0,Y 178.518,Z 350.87,A -85,B 0,C 180,E1 -22650.004,E2 -22650.004} C_VEL
LIN {X 0,Y 178.529,Z 350.869,A -85,B 0,C 180,E1 -22654.874,E2 -22654.874} C_VEL
LIN {X 0,Y 178.633,Z 350.86,A -85,B 0,C 180,E1 -22660.768,E2 -22660.768} C_VEL
LIN {X 0,Y 178.669,Z 350.85,A -85,B 0,C 180,E1 -22664.017,E2 -22664.017} C_VEL
LIN {X 0,Y 178.889,Z 350.826,A -85,B 0,C 180,E1 -22669.152,E2 -22669.152} C_VEL
LIN {X 0,Y 178.928,Z 350.816,A -85,B 0,C 180,E1 -22673.232,E2 -22673.232} C_VEL
LIN {X 0,Y 179.149,Z 350.793,A -85,B 0,C 180,E1 -22677.751,E2 -22677.751} C_VEL
LIN {X 0,Y 179.364,Z 350.767,A -85,B 0,C 180,E1 -22679.999,E2 -22679.999} C_VEL
LIN {X 0,Y 178.871,Z 350.83,A -85,B 0,C 180,E1 -22684.506,E2 -22684.506} C_VEL
LIN {X 0,Y 178.971,Z 350.813,A -85,B 0,C 180,E1 -22689.037,E2 -22689.037} C_VEL
LIN {X 0,Y 178.681,Z 350.851,A -85,B 0,C 180,E1 -22693.65,E2 -22693.65} C_VEL
LIN {X 0,Y 178.643,Z 350.853,A -85,B 0,C 180,E1 -22698.344,E2 -22698.344} C_VEL
LIN {X 0,Y 178.504,Z 350.873,A -85,B 0,C 180,E1 -22703.185,E2 -22703.185} C_VEL
LIN {X 0,Y 178.481,Z 350.875,A -85,B 0,C 180,E1 -22708.197,E2 -22708.197} C_VEL
LIN {X 0,Y 178.679,Z 351.026,A -85,B 0,C 180,E1 -22713.663,E2 -22713.663} C_VEL
LIN {X 0,Y 179.876,Z 357.092,A -85,B 0,C 180,E1 -22718.692,E2 -22718.692} C_VEL
LIN {X 0,Y 181.721,Z 365.202,A -85,B 0,C 180,E1 -22725.075,E2 -22725.075} C_VEL
LIN {X 0,Y 182.53,Z 369.23,A -85,B 0,C 180,E1 -22728.142,E2 -22728.142} C_VEL
LIN {X 0,Y 181.34,Z 373.983,A -85,B 0,C 180,E1 -22731.68,E2 -22731.68} C_VEL
LIN {X 0,Y 179.828,Z 380.456,A -85,B 0,C 180,E1 -22736.441,E2 -22736.441} C_VEL
LIN {X 0,Y 179.75,Z 384.297,A -85,B 0,C 180,E1 -22736.906,E2 -22736.906} C_VEL
LIN {X 0,Y 179.784,Z 398.462,A -85,B 0,C 180,E1 -22738.417,E2 -22738.417} C_VEL
LIN {X 0,Y 180.294,Z 413.824,A -85,B 0,C 180,E1 -22740.522,E2 -22740.522} C_VEL
LIN {X 0,Y 180.931,Z 427.731,A -85,B 0,C 180,E1 -22742.863,E2 -22742.863} C_VEL
LIN {X 0,Y 181.797,Z 441.847,A -85,B 0,C 180,E1 -22745.751,E2 -22745.751} C_VEL
LIN {X 0,Y 182.572,Z 451.808,A -85,B 0,C 180,E1 -22748.132,E2 -22748.132} C_VEL
LIN {X 0,Y 181.134,Z 462.713,A -85,B 0,C 180,E1 -22751.333,E2 -22751.333} C_VEL
LIN {X 0,Y 180.086,Z 472.233,A -85,B 0,C 180,E1 -22754.729,E2 -22754.729} C_VEL
LIN {X 0,Y 179.603,Z 481.382,A -85,B 0,C 180,E1 -22758.719,E2 -22758.719} C_VEL
LIN {X 0,Y 179.853,Z 487.795,A -85,B 0,C 180,E1 -22762.141,E2 -22762.141} C_VEL
LIN {X 0,Y 180.415,Z 492.958,A -85,B 0,C 180,E1 -22765.534,E2 -22765.534} C_VEL
LIN {X 0,Y 180.968,Z 496.952,A -85,B 0,C 180,E1 -22768.889,E2 -22768.889} C_VEL
LIN {X 0,Y 181.138,Z 498.031,A -85,B 0,C 180,E1 -22770.002,E2 -22770.002} C_VEL
LIN {X 0,Y 180.345,Z 499.493,A -85,B 0,C 180,E1 -22772.235,E2 -22772.235} C_VEL
LIN {X 0,Y 179.488,Z 500.554,A -85,B 0,C 180,E1 -22774.494,E2 -22774.494} C_VEL
LIN {X 0,Y 178.1,Z 501.729,A -85,B 0,C 180,E1 -22779.419,E2 -22779.419} C_VEL
LIN {X 0,Y 177.929,Z 501.79,A -85,B 0,C 180,E1 -22783.711,E2 -22783.711} C_VEL
LIN {X 0,Y 179.049,Z 500.891,A -85,B 0,C 180,E1 -22788.303,E2 -22788.303} C_VEL
LIN {X 0,Y 180.697,Z 499.664,A -85,B 0,C 180,E1 -22791.531,E2 -22791.531} C_VEL
LIN {X 0,Y 181.335,Z 498.749,A -85,B 0,C 180,E1 -22793.366,E2 -22793.366} C_VEL
LIN {X 0,Y 181.33,Z 495.111,A -85,B 0,C 180,E1 -22798.883,E2 -22798.883} C_VEL
LIN {X 0,Y 182.493,Z 493.748,A -85,B 0,C 180,E1 -22800.65,E2 -22800.65} C_VEL
LIN {X 0,Y 183.178,Z 493.285,A -85,B 0,C 180,E1 -22801.209,E2 -22801.209} C_VEL
LIN {X 0,Y 191.863,Z 488.081,A -85,B 0,C 180,E1 -22806.307,E2 -22806.307} C_VEL
LIN {X 0,Y 201.306,Z 482.352,A -85,B 0,C 180,E1 -22810.233,E2 -22810.233} C_VEL
LIN {X 0,Y 211.951,Z 475.144,A -85,B 0,C 180,E1 -22814.135,E2 -22814.135} C_VEL
LIN {X 0,Y 218.442,Z 470.443,A -85,B 0,C 180,E1 -22816.379,E2 -22816.379} C_VEL
LIN {X 0,Y 225.288,Z 465.095,A -85,B 0,C 180,E1 -22819.073,E2 -22819.073} C_VEL
LIN {X 0,Y 227.378,Z 463.417,A -85,B 0,C 180,E1 -22819.988,E2 -22819.988} C_VEL
LIN {X 0,Y 226.713,Z 463.48,A -85,B 0,C 180,E1 -22820.544,E2 -22820.544} C_VEL
LIN {X 0,Y 215.015,Z 467.576,A -85,B 0,C 180,E1 -22823.96,E2 -22823.96} C_VEL
LIN {X 0,Y 206.535,Z 469.651,A -85,B 0,C 180,E1 -22827.013,E2 -22827.013} C_VEL
LIN {X 0,Y 198.841,Z 470.742,A -85,B 0,C 180,E1 -22830.342,E2 -22830.342} C_VEL
LIN {X 0,Y 191.951,Z 470.876,A -85,B 0,C 180,E1 -22833.937,E2 -22833.937} C_VEL
LIN {X 0,Y 186.119,Z 469.981,A -85,B 0,C 180,E1 -22837.815,E2 -22837.815} C_VEL
LIN {X 0,Y 181.131,Z 468.078,A -85,B 0,C 180,E1 -22841.917,E2 -22841.917} C_VEL
LIN {X 0,Y 177.169,Z 465.104,A -85,B 0,C 180,E1 -22846.231,E2 -22846.231} C_VEL
LIN {X 0,Y 174.177,Z 461.023,A -85,B 0,C 180,E1 -22850.712,E2 -22850.712} C_VEL
LIN {X 0,Y 172.346,Z 455.75,A -85,B 0,C 180,E1 -22855.323,E2 -22855.323} C_VEL
LIN {X 0,Y 171.553,Z 449.175,A -85,B 0,C 180,E1 -22860.001,E2 -22860.001} C_VEL
LIN {X 0,Y 171.242,Z 441.097,A -85,B 0,C 180,E1 -22864.709,E2 -22864.709} C_VEL
LIN {X 0,Y 172.06,Z 431.328,A -85,B 0,C 180,E1 -22869.404,E2 -22869.404} C_VEL
LIN {X 0,Y 173.146,Z 421.196,A -85,B 0,C 180,E1 -22873.412,E2 -22873.412} C_VEL
LIN {X 0,Y 174.614,Z 410.482,A -85,B 0,C 180,E1 -22876.967,E2 -22876.967} C_VEL
LIN {X 0,Y 176.384,Z 398.092,A -85,B 0,C 180,E1 -22880.405,E2 -22880.405} C_VEL
LIN {X 0,Y 178.51,Z 384.946,A -85,B 0,C 180,E1 -22883.42,E2 -22883.42} C_VEL
LIN {X 0,Y 179.046,Z 381.795,A -85,B 0,C 180,E1 -22884.047,E2 -22884.047} C_VEL
LIN {X 0,Y 175.862,Z 368.995,A -85,B 0,C 180,E1 -22886.636,E2 -22886.636} C_VEL
LIN {X 0,Y 172.232,Z 354.758,A -85,B 0,C 180,E1 -22889.136,E2 -22889.136} C_VEL
LIN {X 0,Y 171.584,Z 352.205,A -85,B 0,C 180,E1 -22889.65,E2 -22889.65} C_VEL
LIN {X 0,Y 171.491,Z 351.75,A -85,B 0,C 180,E1 -22890.299,E2 -22890.299} C_VEL
LIN {X 0,Y 171.399,Z 351.759,A -85,B 0,C 180,E1 -22895.034,E2 -22895.034} C_VEL
LIN {X 0,Y 171.364,Z 351.764,A -85,B 0,C 180,E1 -22898.807,E2 -22898.807} C_VEL
LIN {X 0,Y 171.345,Z 351.764,A -85,B 0,C 180,E1 -22904.211,E2 -22904.211} C_VEL
LIN {X 0,Y 171.361,Z 351.764,A -85,B 0,C 180,E1 -22908.987,E2 -22908.987} C_VEL
LIN {X 0,Y 171.421,Z 351.756,A -85,B 0,C 180,E1 -22912.047,E2 -22912.047} C_VEL
LIN {X 0,Y 171.416,Z 351.754,A -85,B 0,C 180,E1 -22915.086,E2 -22915.086} C_VEL
LIN {X 0,Y 171.453,Z 351.75,A -85,B 0,C 180,E1 -22920.533,E2 -22920.533} C_VEL
LIN {X 0,Y 171.451,Z 351.753,A -85,B 0,C 180,E1 -22925.798,E2 -22925.798} C_VEL
LIN {X 0,Y 171.584,Z 351.731,A -85,B 0,C 180,E1 -22930.87,E2 -22930.87} C_VEL
LIN {X 0,Y 171.615,Z 351.734,A -85,B 0,C 180,E1 -22935.774,E2 -22935.774} C_VEL
LIN {X 0,Y 171.915,Z 351.692,A -85,B 0,C 180,E1 -22940.587,E2 -22940.587} C_VEL
LIN {X 0,Y 171.83,Z 351.705,A -85,B 0,C 180,E1 -22945.306,E2 -22945.306} C_VEL
LIN {X 0,Y 172.337,Z 351.643,A -85,B 0,C 180,E1 -22949.998,E2 -22949.998} C_VEL
LIN {X 0,Y 171.83,Z 351.703,A -85,B 0,C 180,E1 -22954.69,E2 -22954.69} C_VEL
LIN {X 0,Y 171.913,Z 351.695,A -85,B 0,C 180,E1 -22959.409,E2 -22959.409} C_VEL
LIN {X 0,Y 171.615,Z 351.727,A -85,B 0,C 180,E1 -22964.222,E2 -22964.222} C_VEL
LIN {X 0,Y 171.559,Z 351.741,A -85,B 0,C 180,E1 -22969.572,E2 -22969.572} C_VEL
LIN {X 0,Y 171.469,Z 351.751,A -85,B 0,C 180,E1 -22975.614,E2 -22975.614} C_VEL
LIN {X 0,Y 171.439,Z 351.752,A -85,B 0,C 180,E1 -22980.583,E2 -22980.583} C_VEL
LIN {X 0,Y 171.391,Z 351.76,A -85,B 0,C 180,E1 -22985.032,E2 -22985.032} C_VEL
LIN {X 0,Y 171.356,Z 351.764,A -85,B 0,C 180,E1 -22988.805,E2 -22988.805} C_VEL
LIN {X 0,Y 171.321,Z 351.768,A -85,B 0,C 180,E1 -22994.214,E2 -22994.214} C_VEL
LIN {X 0,Y 171.335,Z 351.764,A -85,B 0,C 180,E1 -22998.98,E2 -22998.98} C_VEL
LIN {X 0,Y 171.383,Z 351.76,A -85,B 0,C 180,E1 -23002.039,E2 -23002.039} C_VEL
LIN {X 0,Y 171.394,Z 351.759,A -85,B 0,C 180,E1 -23005.09,E2 -23005.09} C_VEL
LIN {X 0,Y 171.445,Z 351.753,A -85,B 0,C 180,E1 -23010.533,E2 -23010.533} C_VEL
LIN {X 0,Y 171.454,Z 351.747,A -85,B 0,C 180,E1 -23015.8,E2 -23015.8} C_VEL
LIN {X 0,Y 171.59,Z 351.736,A -85,B 0,C 180,E1 -23020.872,E2 -23020.872} C_VEL
LIN {X 0,Y 171.607,Z 351.729,A -85,B 0,C 180,E1 -23025.775,E2 -23025.775} C_VEL
LIN {X 0,Y 171.904,Z 351.697,A -85,B 0,C 180,E1 -23030.587,E2 -23030.587} C_VEL
LIN {X 0,Y 171.82,Z 351.705,A -85,B 0,C 180,E1 -23035.307,E2 -23035.307} C_VEL
LIN {X 0,Y 172.327,Z 351.643,A -85,B 0,C 180,E1 -23039.999,E2 -23039.999} C_VEL
LIN {X 0,Y 171.82,Z 351.707,A -85,B 0,C 180,E1 -23044.692,E2 -23044.692} C_VEL
LIN {X 0,Y 171.903,Z 351.693,A -85,B 0,C 180,E1 -23049.411,E2 -23049.411} C_VEL
LIN {X 0,Y 171.603,Z 351.736,A -85,B 0,C 180,E1 -23054.224,E2 -23054.224} C_VEL
LIN {X 0,Y 171.538,Z 351.737,A -85,B 0,C 180,E1 -23059.562,E2 -23059.562} C_VEL
LIN {X 0,Y 171.463,Z 351.751,A -85,B 0,C 180,E1 -23065.617,E2 -23065.617} C_VEL
LIN {X 0,Y 171.472,Z 351.749,A -85,B 0,C 180,E1 -23070.608,E2 -23070.608} C_VEL
LIN {X 0,Y 171.641,Z 351.932,A -85,B 0,C 180,E1 -23073.733,E2 -23073.733} C_VEL
LIN {X 0,Y 172.987,Z 358.637,A -85,B 0,C 180,E1 -23079.477,E2 -23079.477} C_VEL
LIN {X 0,Y 174.52,Z 365.15,A -85,B 0,C 180,E1 -23084.806,E2 -23084.806} C_VEL
LIN {X 0,Y 175.363,Z 368.958,A -85,B 0,C 180,E1 -23087.823,E2 -23087.823} C_VEL
LIN {X 0,Y 174.848,Z 371.721,A -85,B 0,C 180,E1 -23089.978,E2 -23089.978} C_VEL
LIN {X 0,Y 172.859,Z 379.582,A -85,B 0,C 180,E1 -23096.013,E2 -23096.013} C_VEL
LIN {X 0,Y 172.702,Z 397.602,A -85,B 0,C 180,E1 -23098.063,E2 -23098.063} C_VEL
LIN {X 0,Y 173.207,Z 413.581,A -85,B 0,C 180,E1 -23100.365,E2 -23100.365} C_VEL
LIN {X 0,Y 173.855,Z 428.24,A -85,B 0,C 180,E1 -23102.995,E2 -23102.995} C_VEL
LIN {X 0,Y 174.748,Z 441.98,A -85,B 0,C 180,E1 -23105.973,E2 -23105.973} C_VEL
LIN {X 0,Y 175.467,Z 451.449,A -85,B 0,C 180,E1 -23108.371,E2 -23108.371} C_VEL
LIN {X 0,Y 174.031,Z 462.335,A -85,B 0,C 180,E1 -23111.764,E2 -23111.764} C_VEL
LIN {X 0,Y 173.104,Z 471.702,A -85,B 0,C 180,E1 -23115.303,E2 -23115.303} C_VEL
LIN {X 0,Y 172.786,Z 480.682,A -85,B 0,C 180,E1 -23119.456,E2 -23119.456} C_VEL
LIN {X 0,Y 173.111,Z 486.944,A -85,B 0,C 180,E1 -23123.006,E2 -23123.006} C_VEL
LIN {X 0,Y 173.769,Z 491.972,A -85,B 0,C 180,E1 -23126.524,E2 -23126.524} C_VEL
LIN {X 0,Y 174.346,Z 495.804,A -85,B 0,C 180,E1 -23130.002,E2 -23130.002} C_VEL
LIN {X 0,Y 173.516,Z 497.377,A -85,B 0,C 180,E1 -23132.323,E2 -23132.323} C_VEL
LIN {X 0,Y 171.814,Z 499.35,A -85,B 0,C 180,E1 -23137.051,E2 -23137.051} C_VEL
LIN {X 0,Y 170.995,Z 500.104,A -85,B 0,C 180,E1 -23141.861,E2 -23141.861} C_VEL
LIN {X 0,Y 171.514,Z 499.912,A -85,B 0,C 180,E1 -23146.671,E2 -23146.671} C_VEL
LIN {X 0,Y 173.802,Z 498.631,A -85,B 0,C 180,E1 -23151.954,E2 -23151.954} C_VEL
LIN {X 0,Y 179.092,Z 495.597,A -85,B 0,C 180,E1 -23158.095,E2 -23158.095} C_VEL
LIN {X 0,Y 183.178,Z 493.285,A -85,B 0,C 180,E1 -23161.209,E2 -23161.209} C_VEL
LIN {X 0,Y 184.985,Z 491.879,A -85,B 0,C 180,E1 -23162.907,E2 -23162.907} C_VEL
LIN {X 0,Y 188.595,Z 487.218,A -85,B 0,C 180,E1 -23168.069,E2 -23168.069} C_VEL
LIN {X 0,Y 190.948,Z 485.432,A -85,B 0,C 180,E1 -23169.6,E2 -23169.6} C_VEL
LIN {X 0,Y 192.009,Z 484.81,A -85,B 0,C 180,E1 -23170.055,E2 -23170.055} C_VEL
LIN {X 0,Y 204.646,Z 477.357,A -85,B 0,C 180,E1 -23174.752,E2 -23174.752} C_VEL
LIN {X 0,Y 211.499,Z 473.027,A -85,B 0,C 180,E1 -23176.976,E2 -23176.976} C_VEL
LIN {X 0,Y 217.701,Z 468.756,A -85,B 0,C 180,E1 -23179.269,E2 -23179.269} C_VEL
LIN {X 0,Y 219.268,Z 467.478,A -85,B 0,C 180,E1 -23180.131,E2 -23180.131} C_VEL
LIN {X 0,Y 209.695,Z 470.183,A -85,B 0,C 180,E1 -23182.896,E2 -23182.896} C_VEL
LIN {X 0,Y 200.901,Z 471.869,A -85,B 0,C 180,E1 -23185.964,E2 -23185.964} C_VEL
LIN {X 0,Y 192.929,Z 472.603,A -85,B 0,C 180,E1 -23189.337,E2 -23189.337} C_VEL
LIN {X 0,Y 185.747,Z 472.396,A -85,B 0,C 180,E1 -23192.997,E2 -23192.997} C_VEL
LIN {X 0,Y 179.683,Z 471.171,A -85,B 0,C 180,E1 -23196.975,E2 -23196.975} C_VEL
LIN {X 0,Y 174.453,Z 468.939,A -85,B 0,C 180,E1 -23201.199,E2 -23201.199} C_VEL
LIN {X 0,Y 170.302,Z 465.634,A -85,B 0,C 180,E1 -23205.665,E2 -23205.665} C_VEL
LIN {X 0,Y 167.18,Z 461.234,A -85,B 0,C 180,E1 -23210.32,E2 -23210.32} C_VEL
LIN {X 0,Y 165.283,Z 455.652,A -85,B 0,C 180,E1 -23215.122,E2 -23215.122} C_VEL
LIN {X 0,Y 164.473,Z 448.775,A -85,B 0,C 180,E1 -23220.001,E2 -23220.001} C_VEL
LIN {X 0,Y 164.148,Z 440.34,A -85,B 0,C 180,E1 -23224.913,E2 -23224.913} C_VEL
LIN {X 0,Y 165.076,Z 430.019,A -85,B 0,C 180,E1 -23229.863,E2 -23229.863} C_VEL
LIN {X 0,Y 166.227,Z 419.404,A -85,B 0,C 180,E1 -23234.07,E2 -23234.07} C_VEL
LIN {X 0,Y 167.924,Z 407.543,A -85,B 0,C 180,E1 -23237.979,E2 -23237.979} C_VEL
LIN {X 0,Y 169.93,Z 394.412,A -85,B 0,C 180,E1 -23241.535,E2 -23241.535} C_VEL
LIN {X 0,Y 171.848,Z 381.926,A -85,B 0,C 180,E1 -23244.347,E2 -23244.347} C_VEL
LIN {X 0,Y 168.575,Z 369.135,A -85,B 0,C 180,E1 -23247.015,E2 -23247.015} C_VEL
LIN {X 0,Y 164.563,Z 353.201,A -85,B 0,C 180,E1 -23249.955,E2 -23249.955} C_VEL
LIN {X 0,Y 164.474,Z 352.662,A -85,B 0,C 180,E1 -23250.352,E2 -23250.352} C_VEL
LIN {X 0,Y 164.336,Z 352.638,A -85,B 0,C 180,E1 -23255.651,E2 -23255.651} C_VEL
LIN {X 0,Y 164.298,Z 352.643,A -85,B 0,C 180,E1 -23259.915,E2 -23259.915} C_VEL
LIN {X 0,Y 164.285,Z 352.643,A -85,B 0,C 180,E1 -23263.341,E2 -23263.341} C_VEL
LIN {X 0,Y 164.298,Z 352.643,A -85,B 0,C 180,E1 -23266.808,E2 -23266.808} C_VEL
LIN {X 0,Y 164.315,Z 352.643,A -85,B 0,C 180,E1 -23270.345,E2 -23270.345} C_VEL
LIN {X 0,Y 164.349,Z 352.634,A -85,B 0,C 180,E1 -23274.341,E2 -23274.341} C_VEL
LIN {X 0,Y 164.395,Z 352.631,A -85,B 0,C 180,E1 -23279.133,E2 -23279.133} C_VEL
LIN {X 0,Y 164.412,Z 352.629,A -85,B 0,C 180,E1 -23284.691,E2 -23284.691} C_VEL
LIN {X 0,Y 164.49,Z 352.616,A -85,B 0,C 180,E1 -23290.05,E2 -23290.05} C_VEL
LIN {X 0,Y 164.559,Z 352.611,A -85,B 0,C 180,E1 -23295.15,E2 -23295.15} C_VEL
LIN {X 0,Y 164.858,Z 352.572,A -85,B 0,C 180,E1 -23300.18,E2 -23300.18} C_VEL
LIN {X 0,Y 164.867,Z 352.572,A -85,B 0,C 180,E1 -23302.65,E2 -23302.65} C_VEL
LIN {X 0,Y 165.055,Z 352.546,A -85,B 0,C 180,E1 -23307.557,E2 -23307.557} C_VEL
LIN {X 0,Y 165.3,Z 352.519,A -85,B 0,C 180,E1 -23309.998,E2 -23309.998} C_VEL
LIN {X 0,Y 164.78,Z 352.581,A -85,B 0,C 180,E1 -23314.891,E2 -23314.891} C_VEL
LIN {X 0,Y 164.866,Z 352.569,A -85,B 0,C 180,E1 -23317.345,E2 -23317.345} C_VEL
LIN {X 0,Y 164.782,Z 352.584,A -85,B 0,C 180,E1 -23321.196,E2 -23321.196} C_VEL
LIN {X 0,Y 164.522,Z 352.615,A -85,B 0,C 180,E1 -23327.397,E2 -23327.397} C_VEL
LIN {X 0,Y 164.476,Z 352.621,A -85,B 0,C 180,E1 -23329.986,E2 -23329.986} C_VEL
LIN {X 0,Y 164.393,Z 352.631,A -85,B 0,C 180,E1 -23336.131,E2 -23336.131} C_VEL
LIN {X 0,Y 164.373,Z 352.631,A -85,B 0,C 180,E1 -23341.224,E2 -23341.224} C_VEL
LIN {X 0,Y 164.293,Z 352.645,A -85,B 0,C 180,E1 -23346.787,E2 -23346.787} C_VEL
LIN {X 0,Y 164.29,Z 352.64,A -85,B 0,C 180,E1 -23349.913,E2 -23349.913} C_VEL
LIN {X 0,Y 164.276,Z 352.647,A -85,B 0,C 180,E1 -23353.339,E2 -23353.339} C_VEL
LIN {X 0,Y 164.289,Z 352.646,A -85,B 0,C 180,E1 -23356.806,E2 -23356.806} C_VEL
LIN {X 0,Y 164.292,Z 352.64,A -85,B 0,C 180,E1 -23360.349,E2 -23360.349} C_VEL
LIN {X 0,Y 164.325,Z 352.638,A -85,B 0,C 180,E1 -23366.22,E2 -23366.22} C_VEL
LIN {X 0,Y 164.401,Z 352.63,A -85,B 0,C 180,E1 -23369.136,E2 -23369.136} C_VEL
LIN {X 0,Y 164.412,Z 352.628,A -85,B 0,C 180,E1 -23374.692,E2 -23374.692} C_VEL
LIN {X 0,Y 164.481,Z 352.621,A -85,B 0,C 180,E1 -23380.048,E2 -23380.048} C_VEL
LIN {X 0,Y 164.553,Z 352.608,A -85,B 0,C 180,E1 -23385.151,E2 -23385.151} C_VEL
LIN {X 0,Y 164.847,Z 352.576,A -85,B 0,C 180,E1 -23390.18,E2 -23390.18} C_VEL
LIN {X 0,Y 164.856,Z 352.57,A -85,B 0,C 180,E1 -23392.651,E2 -23392.651} C_VEL
LIN {X 0,Y 165.045,Z 352.55,A -85,B 0,C 180,E1 -23397.559,E2 -23397.559} C_VEL
LIN {X 0,Y 165.289,Z 352.52,A -85,B 0,C 180,E1 -23399.999,E2 -23399.999} C_VEL
LIN {X 0,Y 164.77,Z 352.585,A -85,B 0,C 180,E1 -23404.893,E2 -23404.893} C_VEL
LIN {X 0,Y 164.846,Z 352.573,A -85,B 0,C 180,E1 -23409.818,E2 -23409.818} C_VEL
LIN {X 0,Y 164.547,Z 352.612,A -85,B 0,C 180,E1 -23414.848,E2 -23414.848} C_VEL
LIN {X 0,Y 164.467,Z 352.619,A -85,B 0,C 180,E1 -23419.989,E2 -23419.989} C_VEL
LIN {X 0,Y 164.387,Z 352.63,A -85,B 0,C 180,E1 -23426.135,E2 -23426.135} C_VEL
LIN {X 0,Y 164.483,Z 352.621,A -85,B 0,C 180,E1 -23432.373,E2 -23432.373} C_VEL
LIN {X 0,Y 164.589,Z 352.706,A -85,B 0,C 180,E1 -23433.717,E2 -23433.717} C_VEL
LIN {X 0,Y 165.896,Z 359.117,A -85,B 0,C 180,E1 -23439.453,E2 -23439.453} C_VEL
LIN {X 0,Y 167.605,Z 366.171,A -85,B 0,C 180,E1 -23445.466,E2 -23445.466} C_VEL
LIN {X 0,Y 168.259,Z 369.344,A -85,B 0,C 180,E1 -23448.067,E2 -23448.067} C_VEL
LIN {X 0,Y 167.363,Z 372.859,A -85,B 0,C 180,E1 -23450.961,E2 -23450.961} C_VEL
LIN {X 0,Y 165.91,Z 378.729,A -85,B 0,C 180,E1 -23455.584,E2 -23455.584} C_VEL
LIN {X 0,Y 165.618,Z 395.974,A -85,B 0,C 180,E1 -23457.605,E2 -23457.605} C_VEL
LIN {X 0,Y 166.037,Z 411.977,A -85,B 0,C 180,E1 -23460.003,E2 -23460.003} C_VEL
LIN {X 0,Y 166.65,Z 425.746,A -85,B 0,C 180,E1 -23462.543,E2 -23462.543} C_VEL
LIN {X 0,Y 167.483,Z 439.769,A -85,B 0,C 180,E1 -23465.678,E2 -23465.678} C_VEL
LIN {X 0,Y 168.404,Z 450.817,A -85,B 0,C 180,E1 -23468.585,E2 -23468.585} C_VEL
LIN {X 0,Y 166.967,Z 461.861,A -85,B 0,C 180,E1 -23472.234,E2 -23472.234} C_VEL
LIN {X 0,Y 166.157,Z 471.326,A -85,B 0,C 180,E1 -23476.036,E2 -23476.036} C_VEL
LIN {X 0,Y 166.014,Z 479.887,A -85,B 0,C 180,E1 -23480.253,E2 -23480.253} C_VEL
LIN {X 0,Y 166.434,Z 486.021,A -85,B 0,C 180,E1 -23483.942,E2 -23483.942} C_VEL
LIN {X 0,Y 167.172,Z 490.913,A -85,B 0,C 180,E1 -23487.593,E2 -23487.593} C_VEL
LIN {X 0,Y 167.547,Z 493.477,A -85,B 0,C 180,E1 -23490.002,E2 -23490.002} C_VEL
LIN {X 0,Y 166.716,Z 495.164,A -85,B 0,C 180,E1 -23492.418,E2 -23492.418} C_VEL
LIN {X 0,Y 164.942,Z 497.283,A -85,B 0,C 180,E1 -23497.346,E2 -23497.346} C_VEL
LIN {X 0,Y 164.152,Z 498.276,A -85,B 0,C 180,E1 -23502.363,E2 -23502.363} C_VEL
LIN {X 0,Y 164.75,Z 498.295,A -85,B 0,C 180,E1 -23507.376,E2 -23507.376} C_VEL
LIN {X 0,Y 166.863,Z 497.448,A -85,B 0,C 180,E1 -23512.278,E2 -23512.278} C_VEL
LIN {X 0,Y 170.482,Z 495.809,A -85,B 0,C 180,E1 -23516.968,E2 -23516.968} C_VEL
LIN {X 0,Y 176.692,Z 492.794,A -85,B 0,C 180,E1 -23522.097,E2 -23522.097} C_VEL
LIN {X 0,Y 185.762,Z 488.097,A -85,B 0,C 180,E1 -23527.393,E2 -23527.393} C_VEL
LIN {X 0,Y 192.009,Z 484.81,A -85,B 0,C 180,E1 -23530.055,E2 -23530.055} C_VEL
LIN {X 0,Y 194.928,Z 482.962,A -85,B 0,C 180,E1 -23531.465,E2 -23531.465} C_VEL
LIN {X 0,Y 198.395,Z 480.017,A -85,B 0,C 180,E1 -23534.02,E2 -23534.02} C_VEL
LIN {X 0,Y 201.151,Z 477.592,A -85,B 0,C 180,E1 -23536.051,E2 -23536.051} C_VEL
LIN {X 0,Y 203.895,Z 475.613,A -85,B 0,C 180,E1 -23537.433,E2 -23537.433} C_VEL
LIN {X 0,Y 205.016,Z 474.911,A -85,B 0,C 180,E1 -23537.846,E2 -23537.846} C_VEL
LIN {X 0,Y 209.805,Z 472.009,A -85,B 0,C 180,E1 -23539.493,E2 -23539.493} C_VEL
LIN {X 0,Y 210.247,Z 471.469,A -85,B 0,C 180,E1 -23540.085,E2 -23540.085} C_VEL
LIN {X 0,Y 199.771,Z 473.493,A -85,B 0,C 180,E1 -23543.269,E2 -23543.269} C_VEL
LIN {X 0,Y 191.108,Z 474.322,A -85,B 0,C 180,E1 -23546.522,E2 -23546.522} C_VEL
LIN {X 0,Y 183.21,Z 474.213,A -85,B 0,C 180,E1 -23550.088,E2 -23550.088} C_VEL
LIN {X 0,Y 176.319,Z 473.117,A -85,B 0,C 180,E1 -23553.995,E2 -23553.995} C_VEL
LIN {X 0,Y 170.393,Z 471.043,A -85,B 0,C 180,E1 -23558.21,E2 -23558.21} C_VEL
LIN {X 0,Y 165.53,Z 467.949,A -85,B 0,C 180,E1 -23562.711,E2 -23562.711} C_VEL
LIN {X 0,Y 161.668,Z 463.8,A -85,B 0,C 180,E1 -23567.447,E2 -23567.447} C_VEL
LIN {X 0,Y 159.063,Z 458.508,A -85,B 0,C 180,E1 -23572.384,E2 -23572.384} C_VEL
LIN {X 0,Y 157.652,Z 451.968,A -85,B 0,C 180,E1 -23577.446,E2 -23577.446} C_VEL
LIN {X 0,Y 157.217,Z 445.095,A -85,B 0,C 180,E1 -23581.922,E2 -23581.922} C_VEL
LIN {X 0,Y 157.306,Z 435.653,A -85,B 0,C 180,E1 -23587.058,E2 -23587.058} C_VEL
LIN {X 0,Y 158.184,Z 427.47,A -85,B 0,C 180,E1 -23590.826,E2 -23590.826} C_VEL
LIN {X 0,Y 159.593,Z 415.894,A -85,B 0,C 180,E1 -23595.321,E2 -23595.321} C_VEL
LIN {X 0,Y 161.316,Z 404.253,A -85,B 0,C 180,E1 -23599.072,E2 -23599.072} C_VEL
LIN {X 0,Y 163.556,Z 390.364,A -85,B 0,C 180,E1 -23602.752,E2 -23602.752} C_VEL
LIN {X 0,Y 164.616,Z 383.709,A -85,B 0,C 180,E1 -23604.264,E2 -23604.264} C_VEL
LIN {X 0,Y 164.332,Z 381.205,A -85,B 0,C 180,E1 -23604.837,E2 -23604.837} C_VEL
LIN {X 0,Y 160.747,Z 367.136,A -85,B 0,C 180,E1 -23607.805,E2 -23607.805} C_VEL
LIN {X 0,Y 157.621,Z 354.524,A -85,B 0,C 180,E1 -23610.137,E2 -23610.137} C_VEL
LIN {X 0,Y 157.415,Z 353.538,A -85,B 0,C 180,E1 -23610.707,E2 -23610.707} C_VEL
LIN {X 0,Y 157.274,Z 353.516,A -85,B 0,C 180,E1 -23616.449,E2 -23616.449} C_VEL
LIN {X 0,Y 157.217,Z 353.526,A -85,B 0,C 180,E1 -23622.11,E2 -23622.11} C_VEL
LIN {X 0,Y 157.22,Z 353.524,A -85,B 0,C 180,E1 -23627.89,E2 -23627.89} C_VEL
LIN {X 0,Y 157.289,Z 353.511,A -85,B 0,C 180,E1 -23633.542,E2 -23633.542} C_VEL
LIN {X 0,Y 157.299,Z 353.517,A -85,B 0,C 180,E1 -23638.094,E2 -23638.094} C_VEL
LIN {X 0,Y 157.32,Z 353.509,A -85,B 0,C 180,E1 -23643.463,E2 -23643.463} C_VEL
LIN {X 0,Y 157.398,Z 353.501,A -85,B 0,C 180,E1 -23649.667,E2 -23649.667} C_VEL
LIN {X 0,Y 157.484,Z 353.493,A -85,B 0,C 180,E1 -23654.467,E2 -23654.467} C_VEL
LIN {X 0,Y 157.777,Z 353.451,A -85,B 0,C 180,E1 -23659.734,E2 -23659.734} C_VEL
LIN {X 0,Y 157.829,Z 353.45,A -85,B 0,C 180,E1 -23662.321,E2 -23662.321} C_VEL
LIN {X 0,Y 158.262,Z 353.396,A -85,B 0,C 180,E1 -23669.998,E2 -23669.998} C_VEL
LIN {X 0,Y 157.828,Z 353.447,A -85,B 0,C 180,E1 -23677.675,E2 -23677.675} C_VEL
LIN {X 0,Y 157.708,Z 353.466,A -85,B 0,C 180,E1 -23681.36,E2 -23681.36} C_VEL
LIN {X 0,Y 157.487,Z 353.488,A -85,B 0,C 180,E1 -23685.528,E2 -23685.528} C_VEL
LIN {X 0,Y 157.372,Z 353.506,A -85,B 0,C 180,E1 -23690.93,E2 -23690.93} C_VEL
LIN {X 0,Y 157.314,Z 353.513,A -85,B 0,C 180,E1 -23696.682,E2 -23696.682} C_VEL
LIN {X 0,Y 157.273,Z 353.513,A -85,B 0,C 180,E1 -23702.425,E2 -23702.425} C_VEL
LIN {X 0,Y 157.266,Z 353.519,A -85,B 0,C 180,E1 -23706.447,E2 -23706.447} C_VEL
LIN {X 0,Y 157.208,Z 353.524,A -85,B 0,C 180,E1 -23712.108,E2 -23712.108} C_VEL
LIN {X 0,Y 157.207,Z 353.523,A -85,B 0,C 180,E1 -23717.887,E2 -23717.887} C_VEL
LIN {X 0,Y 157.264,Z 353.52,A -85,B 0,C 180,E1 -23723.548,E2 -23723.548} C_VEL
LIN {X 0,Y 157.297,Z 353.51,A -85,B 0,C 180,E1 -23728.089,E2 -23728.089} C_VEL
LIN {X 0,Y 157.317,Z 353.512,A -85,B 0,C 180,E1 -23733.464,E2 -23733.464} C_VEL
LIN {X 0,Y 157.39,Z 353.503,A -85,B 0,C 180,E1 -23739.664,E2 -23739.664} C_VEL
LIN {X 0,Y 157.48,Z 353.489,A -85,B 0,C 180,E1 -23744.468,E2 -23744.468} C_VEL
LIN {X 0,Y 157.766,Z 353.457,A -85,B 0,C 180,E1 -23749.735,E2 -23749.735} C_VEL
LIN {X 0,Y 157.818,Z 353.448,A -85,B 0,C 180,E1 -23752.322,E2 -23752.322} C_VEL
LIN {X 0,Y 158.252,Z 353.396,A -85,B 0,C 180,E1 -23759.999,E2 -23759.999} C_VEL
LIN {X 0,Y 157.818,Z 353.451,A -85,B 0,C 180,E1 -23767.677,E2 -23767.677} C_VEL
LIN {X 0,Y 157.699,Z 353.461,A -85,B 0,C 180,E1 -23771.362,E2 -23771.362} C_VEL
LIN {X 0,Y 157.472,Z 353.494,A -85,B 0,C 180,E1 -23775.532,E2 -23775.532} C_VEL
LIN {X 0,Y 157.363,Z 353.505,A -85,B 0,C 180,E1 -23780.933,E2 -23780.933} C_VEL
LIN {X 0,Y 157.309,Z 353.509,A -85,B 0,C 180,E1 -23786.686,E2 -23786.686} C_VEL
LIN {X 0,Y 157.567,Z 353.599,A -85,B 0,C 180,E1 -23793.885,E2 -23793.885} C_VEL
LIN {X 0,Y 158.917,Z 360.021,A -85,B 0,C 180,E1 -23799.869,E2 -23799.869} C_VEL
LIN {X 0,Y 160.506,Z 366.394,A -85,B 0,C 180,E1 -23805.53,E2 -23805.53} C_VEL
LIN {X 0,Y 161.093,Z 369.122,A -85,B 0,C 180,E1 -23807.872,E2 -23807.872} C_VEL
LIN {X 0,Y 160.367,Z 372.229,A -85,B 0,C 180,E1 -23810.55,E2 -23810.55} C_VEL
LIN {X 0,Y 158.933,Z 377.639,A -85,B 0,C 180,E1 -23815.088,E2 -23815.088} C_VEL
LIN {X 0,Y 158.573,Z 395.806,A -85,B 0,C 180,E1 -23817.36,E2 -23817.36} C_VEL
LIN {X 0,Y 158.891,Z 411.189,A -85,B 0,C 180,E1 -23819.795,E2 -23819.795} C_VEL
LIN {X 0,Y 159.559,Z 425.311,A -85,B 0,C 180,E1 -23822.548,E2 -23822.548} C_VEL
LIN {X 0,Y 160.412,Z 439.45,A -85,B 0,C 180,E1 -23825.886,E2 -23825.886} C_VEL
LIN {X 0,Y 161.378,Z 449.354,A -85,B 0,C 180,E1 -23828.612,E2 -23828.612} C_VEL
LIN {X 0,Y 160.142,Z 459.605,A -85,B 0,C 180,E1 -23832.112,E2 -23832.112} C_VEL
LIN {X 0,Y 159.294,Z 469.833,A -85,B 0,C 180,E1 -23836.376,E2 -23836.376} C_VEL
LIN {X 0,Y 159.185,Z 477.878,A -85,B 0,C 180,E1 -23840.473,E2 -23840.473} C_VEL
LIN {X 0,Y 159.809,Z 485.013,A -85,B 0,C 180,E1 -23844.956,E2 -23844.956} C_VEL
LIN {X 0,Y 160.572,Z 489.755,A -85,B 0,C 180,E1 -23848.748,E2 -23848.748} C_VEL
LIN {X 0,Y 160.771,Z 491.046,A -85,B 0,C 180,E1 -23850.002,E2 -23850.002} C_VEL
LIN {X 0,Y 159.961,Z 492.855,A -85,B 0,C 180,E1 -23852.52,E2 -23852.52} C_VEL
LIN {X 0,Y 158.093,Z 495.177,A -85,B 0,C 180,E1 -23857.666,E2 -23857.666} C_VEL
LIN {X 0,Y 157.358,Z 496.325,A -85,B 0,C 180,E1 -23862.906,E2 -23862.906} C_VEL
LIN {X 0,Y 158.045,Z 496.575,A -85,B 0,C 180,E1 -23868.139,E2 -23868.139} C_VEL
LIN {X 0,Y 160.359,Z 495.981,A -85,B 0,C 180,E1 -23873.233,E2 -23873.233} C_VEL
LIN {X 0,Y 164.19,Z 494.593,A -85,B 0,C 180,E1 -23878.091,E2 -23878.091} C_VEL
LIN {X 0,Y 169.619,Z 492.463,A -85,B 0,C 180,E1 -23882.594,E2 -23882.594} C_VEL
LIN {X 0,Y 179.578,Z 488.015,A -85,B 0,C 180,E1 -23888.49,E2 -23888.49} C_VEL
LIN {X 0,Y 190.676,Z 482.739,A -85,B 0,C 180,E1 -23892.993,E2 -23892.993} C_VEL
LIN {X 0,Y 205.016,Z 474.911,A -85,B 0,C 180,E1 -23897.846,E2 -23897.846} C_VEL
LIN {X 0,Y 205.53,Z 474.396,A -85,B 0,C 180,E1 -23898.332,E2 -23898.332} C_VEL
LIN {X 0,Y 204.949,Z 474.157,A -85,B 0,C 180,E1 -23899.028,E2 -23899.028} C_VEL
LIN {X 0,Y 202.863,Z 474.306,A -85,B 0,C 180,E1 -23899.942,E2 -23899.942} C_VEL
LIN {X 0,Y 192.335,Z 475.864,A -85,B 0,C 180,E1 -23902.777,E2 -23902.777} C_VEL
LIN {X 0,Y 181.229,Z 476.011,A -85,B 0,C 180,E1 -23907.118,E2 -23907.118} C_VEL
LIN {X 0,Y 173.458,Z 475.069,A -85,B 0,C 180,E1 -23910.909,E2 -23910.909} C_VEL
LIN {X 0,Y 166.835,Z 473.144,A -85,B 0,C 180,E1 -23915.087,E2 -23915.087} C_VEL
LIN {X 0,Y 161.133,Z 470.246,A -85,B 0,C 180,E1 -23919.579,E2 -23919.579} C_VEL
LIN {X 0,Y 156.601,Z 466.306,A -85,B 0,C 180,E1 -23924.38,E2 -23924.38} C_VEL
LIN {X 0,Y 153.222,Z 461.265,A -85,B 0,C 180,E1 -23929.429,E2 -23929.429} C_VEL
LIN {X 0,Y 151.173,Z 455.042,A -85,B 0,C 180,E1 -23934.666,E2 -23934.666} C_VEL
LIN {X 0,Y 150.32,Z 447.5,A -85,B 0,C 180,E1 -23940.001,E2 -23940.001} C_VEL
LIN {X 0,Y 150.04,Z 438.308,A -85,B 0,C 180,E1 -23945.376,E2 -23945.376} C_VEL
LIN {X 0,Y 150.989,Z 428.273,A -85,B 0,C 180,E1 -23950.292,E2 -23950.292} C_VEL
LIN {X 0,Y 152.208,Z 417.83,A -85,B 0,C 180,E1 -23954.576,E2 -23954.576} C_VEL
LIN {X 0,Y 154.11,Z 404.951,A -85,B 0,C 180,E1 -23958.962,E2 -23958.962} C_VEL
LIN {X 0,Y 156.329,Z 391.033,A -85,B 0,C 180,E1 -23962.815,E2 -23962.815} C_VEL
LIN {X 0,Y 157.561,Z 383.677,A -85,B 0,C 180,E1 -23964.556,E2 -23964.556} C_VEL
LIN {X 0,Y 154.267,Z 370.363,A -85,B 0,C 180,E1 -23967.552,E2 -23967.552} C_VEL
LIN {X 0,Y 150.447,Z 354.9,A -85,B 0,C 180,E1 -23970.656,E2 -23970.656} C_VEL
LIN {X 0,Y 150.345,Z 354.399,A -85,B 0,C 180,E1 -23971.241,E2 -23971.241} C_VEL
LIN {X 0,Y 150.179,Z 354.398,A -85,B 0,C 180,E1 -23977.473,E2 -23977.473} C_VEL
LIN {X 0,Y 150.156,Z 354.405,A -85,B 0,C 180,E1 -23981.504,E2 -23981.504} C_VEL
LIN {X 0,Y 150.149,Z 354.4,A -85,B 0,C 180,E1 -23985.401,E2 -23985.401} C_VEL
LIN {X 0,Y 150.164,Z 354.404,A -85,B 0,C 180,E1 -23989.06,E2 -23989.06} C_VEL
LIN {X 0,Y 150.222,Z 354.392,A -85,B 0,C 180,E1 -23992.688,E2 -23992.688} C_VEL
LIN {X 0,Y 150.224,Z 354.396,A -85,B 0,C 180,E1 -23997.365,E2 -23997.365} C_VEL
LIN {X 0,Y 150.246,Z 354.39,A -85,B 0,C 180,E1 -24002.719,E2 -24002.719} C_VEL
LIN {X 0,Y 150.355,Z 354.378,A -85,B 0,C 180,E1 -24009.207,E2 -24009.207} C_VEL
LIN {X 0,Y 150.388,Z 354.376,A -85,B 0,C 180,E1 -24013.714,E2 -24013.714} C_VEL
LIN {X 0,Y 150.694,Z 354.333,A -85,B 0,C 180,E1 -24019.246,E2 -24019.246} C_VEL
LIN {X 0,Y 150.768,Z 354.329,A -85,B 0,C 180,E1 -24021.959,E2 -24021.959} C_VEL
LIN {X 0,Y 151.223,Z 354.272,A -85,B 0,C 180,E1 -24029.998,E2 -24029.998} C_VEL
LIN {X 0,Y 150.766,Z 354.328,A -85,B 0,C 180,E1 -24038.036,E2 -24038.036} C_VEL
LIN {X 0,Y 150.637,Z 354.347,A -85,B 0,C 180,E1 -24041.544,E2 -24041.544} C_VEL
LIN {X 0,Y 150.393,Z 354.373,A -85,B 0,C 180,E1 -24046.281,E2 -24046.281} C_VEL
LIN {X 0,Y 150.353,Z 354.38,A -85,B 0,C 180,E1 -24050.791,E2 -24050.791} C_VEL
LIN {X 0,Y 150.244,Z 354.396,A -85,B 0,C 180,E1 -24057.279,E2 -24057.279} C_VEL
LIN {X 0,Y 150.213,Z 354.392,A -85,B 0,C 180,E1 -24062.629,E2 -24062.629} C_VEL
LIN {X 0,Y 150.175,Z 354.403,A -85,B 0,C 180,E1 -24067.469,E2 -24067.469} C_VEL
LIN {X 0,Y 150.148,Z 354.403,A -85,B 0,C 180,E1 -24071.502,E2 -24071.502} C_VEL
LIN {X 0,Y 150.123,Z 354.41,A -85,B 0,C 180,E1 -24075.393,E2 -24075.393} C_VEL
LIN {X 0,Y 150.147,Z 354.402,A -85,B 0,C 180,E1 -24079.056,E2 -24079.056} C_VEL
LIN {X 0,Y 150.178,Z 354.403,A -85,B 0,C 180,E1 -24082.704,E2 -24082.704} C_VEL
LIN {X 0,Y 150.216,Z 354.392,A -85,B 0,C 180,E1 -24087.362,E2 -24087.362} C_VEL
LIN {X 0,Y 150.241,Z 354.396,A -85,B 0,C 180,E1 -24092.715,E2 -24092.715} C_VEL
LIN {X 0,Y 150.347,Z 354.382,A -85,B 0,C 180,E1 -24099.205,E2 -24099.205} C_VEL
LIN {X 0,Y 150.385,Z 354.373,A -85,B 0,C 180,E1 -24103.715,E2 -24103.715} C_VEL
LIN {X 0,Y 150.683,Z 354.339,A -85,B 0,C 180,E1 -24109.247,E2 -24109.247} C_VEL
LIN {X 0,Y 150.757,Z 354.329,A -85,B 0,C 180,E1 -24111.96,E2 -24111.96} C_VEL
LIN {X 0,Y 151.212,Z 354.273,A -85,B 0,C 180,E1 -24119.999,E2 -24119.999} C_VEL
LIN {X 0,Y 150.756,Z 354.331,A -85,B 0,C 180,E1 -24128.039,E2 -24128.039} C_VEL
LIN {X 0,Y 150.628,Z 354.342,A -85,B 0,C 180,E1 -24131.545,E2 -24131.545} C_VEL
LIN {X 0,Y 150.376,Z 354.377,A -85,B 0,C 180,E1 -24136.284,E2 -24136.284} C_VEL
LIN {X 0,Y 150.344,Z 354.38,A -85,B 0,C 180,E1 -24140.793,E2 -24140.793} C_VEL
LIN {X 0,Y 150.241,Z 354.39,A -85,B 0,C 180,E1 -24147.285,E2 -24147.285} C_VEL
LIN {X 0,Y 150.538,Z 354.449,A -85,B 0,C 180,E1 -24154.071,E2 -24154.071} C_VEL
LIN {X 0,Y 151.938,Z 360.915,A -85,B 0,C 180,E1 -24160.359,E2 -24160.359} C_VEL
LIN {X 0,Y 153.733,Z 367.796,A -85,B 0,C 180,E1 -24166.71,E2 -24166.71} C_VEL
LIN {X 0,Y 153.866,Z 369.943,A -85,B 0,C 180,E1 -24168.654,E2 -24168.654} C_VEL
LIN {X 0,Y 151.963,Z 376.632,A -85,B 0,C 180,E1 -24174.585,E2 -24174.585} C_VEL
LIN {X 0,Y 151.675,Z 381.163,A -85,B 0,C 180,E1 -24175.217,E2 -24175.217} C_VEL
LIN {X 0,Y 151.5,Z 395.896,A -85,B 0,C 180,E1 -24177.171,E2 -24177.171} C_VEL
LIN {X 0,Y 151.794,Z 410.616,A -85,B 0,C 180,E1 -24179.647,E2 -24179.647} C_VEL
LIN {X 0,Y 152.422,Z 424.666,A -85,B 0,C 180,E1 -24182.546,E2 -24182.546} C_VEL
LIN {X 0,Y 153.202,Z 437.151,A -85,B 0,C 180,E1 -24185.618,E2 -24185.618} C_VEL
LIN {X 0,Y 154.347,Z 448.869,A -85,B 0,C 180,E1 -24188.99,E2 -24188.99} C_VEL
LIN {X 0,Y 153.149,Z 458.943,A -85,B 0,C 180,E1 -24192.648,E2 -24192.648} C_VEL
LIN {X 0,Y 152.465,Z 468.117,A -85,B 0,C 180,E1 -24196.677,E2 -24196.677} C_VEL
LIN {X 0,Y 152.49,Z 476.94,A -85,B 0,C 180,E1 -24201.388,E2 -24201.388} C_VEL
LIN {X 0,Y 153.225,Z 483.919,A -85,B 0,C 180,E1 -24206.057,E2 -24206.057} C_VEL
LIN {X 0,Y 154.031,Z 488.512,A -85,B 0,C 180,E1 -24210.002,E2 -24210.002} C_VEL
LIN {X 0,Y 153.241,Z 490.434,A -85,B 0,C 180,E1 -24212.631,E2 -24212.631} C_VEL
LIN {X 0,Y 151.313,Z 492.913,A -85,B 0,C 180,E1 -24218.012,E2 -24218.012} C_VEL
LIN {X 0,Y 150.573,Z 494.305,A -85,B 0,C 180,E1 -24223.498,E2 -24223.498} C_VEL
LIN {X 0,Y 151.395,Z 494.73,A -85,B 0,C 180,E1 -24228.965,E2 -24228.965} C_VEL
LIN {X 0,Y 153.914,Z 494.41,A -85,B 0,C 180,E1 -24234.267,E2 -24234.267} C_VEL
LIN {X 0,Y 157.989,Z 493.273,A -85,B 0,C 180,E1 -24239.299,E2 -24239.299} C_VEL
LIN {X 0,Y 163.676,Z 491.46,A -85,B 0,C 180,E1 -24243.934,E2 -24243.934} C_VEL
LIN {X 0,Y 173.598,Z 487.672,A -85,B 0,C 180,E1 -24249.718,E2 -24249.718} C_VEL
LIN {X 0,Y 185.537,Z 482.701,A -85,B 0,C 180,E1 -24254.491,E2 -24254.491} C_VEL
LIN {X 0,Y 199.483,Z 475.958,A -85,B 0,C 180,E1 -24259.083,E2 -24259.083} C_VEL
LIN {X 0,Y 200.656,Z 474.922,A -85,B 0,C 180,E1 -24260.149,E2 -24260.149} C_VEL
LIN {X 0,Y 192.335,Z 475.864,A -85,B 0,C 180,E1 -24262.777,E2 -24262.777} C_VEL
LIN {X 0,Y 188.069,Z 476.283,A -85,B 0,C 180,E1 -24264.005,E2 -24264.005} C_VEL
LIN {X 0,Y 179.996,Z 476.902,A -85,B 0,C 180,E1 -24265.789,E2 -24265.789} C_VEL
LIN {X 0,Y 172.16,Z 476.949,A -85,B 0,C 180,E1 -24267.745,E2 -24267.745} C_VEL
LIN {X 0,Y 168.35,Z 476.439,A -85,B 0,C 180,E1 -24269.246,E2 -24269.246} C_VEL
LIN {X 0,Y 160.483,Z 473.945,A -85,B 0,C 180,E1 -24274.029,E2 -24274.029} C_VEL
LIN {X 0,Y 153.255,Z 469.727,A -85,B 0,C 180,E1 -24279.884,E2 -24279.884} C_VEL
LIN {X 0,Y 148.812,Z 465.202,A -85,B 0,C 180,E1 -24284.945,E2 -24284.945} C_VEL
LIN {X 0,Y 145.647,Z 459.552,A -85,B 0,C 180,E1 -24290.278,E2 -24290.278} C_VEL
LIN {X 0,Y 143.799,Z 452.678,A -85,B 0,C 180,E1 -24295.797,E2 -24295.797} C_VEL
LIN {X 0,Y 143.124,Z 444.395,A -85,B 0,C 180,E1 -24301.408,E2 -24301.408} C_VEL
LIN {X 0,Y 143.192,Z 434.379,A -85,B 0,C 180,E1 -24307.049,E2 -24307.049} C_VEL
LIN {X 0,Y 144.105,Z 425.587,A -85,B 0,C 180,E1 -24311.25,E2 -24311.25} C_VEL
LIN {X 0,Y 145.409,Z 415.352,A -85,B 0,C 180,E1 -24315.416,E2 -24315.416} C_VEL
LIN {X 0,Y 147.222,Z 403.352,A -85,B 0,C 180,E1 -24319.522,E2 -24319.522} C_VEL
LIN {X 0,Y 149.348,Z 390.316,A -85,B 0,C 180,E1 -24323.211,E2 -24323.211} C_VEL
LIN {X 0,Y 150.31,Z 383.496,A -85,B 0,C 180,E1 -24324.887,E2 -24324.887} C_VEL
LIN {X 0,Y 146.765,Z 369.602,A -85,B 0,C 180,E1 -24328.087,E2 -24328.087} C_VEL
LIN {X 0,Y 143.445,Z 355.921,A -85,B 0,C 180,E1 -24330.903,E2 -24330.903} C_VEL
LIN {X 0,Y 143.287,Z 355.3,A -85,B 0,C 180,E1 -24331.409,E2 -24331.409} C_VEL
LIN {X 0,Y 143.084,Z 355.283,A -85,B 0,C 180,E1 -24338.193,E2 -24338.193} C_VEL
LIN {X 0,Y 143.068,Z 355.285,A -85,B 0,C 180,E1 -24343.452,E2 -24343.452} C_VEL
LIN {X 0,Y 143.078,Z 355.285,A -85,B 0,C 180,E1 -24347.461,E2 -24347.461} C_VEL
LIN {X 0,Y 143.114,Z 355.281,A -85,B 0,C 180,E1 -24351.789,E2 -24351.789} C_VEL
LIN {X 0,Y 143.191,Z 355.272,A -85,B 0,C 180,E1 -24357.321,E2 -24357.321} C_VEL
LIN {X 0,Y 143.194,Z 355.268,A -85,B 0,C 180,E1 -24362.063,E2 -24362.063} C_VEL
LIN {X 0,Y 143.281,Z 355.259,A -85,B 0,C 180,E1 -24368.745,E2 -24368.745} C_VEL
LIN {X 0,Y 143.322,Z 355.255,A -85,B 0,C 180,E1 -24372.887,E2 -24372.887} C_VEL
LIN {X 0,Y 143.608,Z 355.215,A -85,B 0,C 180,E1 -24378.709,E2 -24378.709} C_VEL
LIN {X 0,Y 143.69,Z 355.209,A -85,B 0,C 180,E1 -24381.56,E2 -24381.56} C_VEL
LIN {X 0,Y 144.181,Z 355.149,A -85,B 0,C 180,E1 -24389.997,E2 -24389.997} C_VEL
LIN {X 0,Y 143.688,Z 355.209,A -85,B 0,C 180,E1 -24398.435,E2 -24398.435} C_VEL
LIN {X 0,Y 143.573,Z 355.225,A -85,B 0,C 180,E1 -24401.755,E2 -24401.755} C_VEL
LIN {X 0,Y 143.325,Z 355.254,A -85,B 0,C 180,E1 -24407.108,E2 -24407.108} C_VEL
LIN {X 0,Y 143.279,Z 355.262,A -85,B 0,C 180,E1 -24411.253,E2 -24411.253} C_VEL
LIN {X 0,Y 143.19,Z 355.273,A -85,B 0,C 180,E1 -24417.934,E2 -24417.934} C_VEL
LIN {X 0,Y 143.163,Z 355.274,A -85,B 0,C 180,E1 -24423.43,E2 -24423.43} C_VEL
LIN {X 0,Y 143.06,Z 355.284,A -85,B 0,C 180,E1 -24429.687,E2 -24429.687} C_VEL
LIN {X 0,Y 143.053,Z 355.291,A -85,B 0,C 180,E1 -24433.452,E2 -24433.452} C_VEL
LIN {X 0,Y 143.062,Z 355.286,A -85,B 0,C 180,E1 -24437.462,E2 -24437.462} C_VEL
LIN {X 0,Y 143.077,Z 355.286,A -85,B 0,C 180,E1 -24441.802,E2 -24441.802} C_VEL
LIN {X 0,Y 143.182,Z 355.268,A -85,B 0,C 180,E1 -24447.32,E2 -24447.32} C_VEL
LIN {X 0,Y 143.188,Z 355.273,A -85,B 0,C 180,E1 -24452.059,E2 -24452.059} C_VEL
LIN {X 0,Y 143.273,Z 355.262,A -85,B 0,C 180,E1 -24458.743,E2 -24458.743} C_VEL
LIN {X 0,Y 143.317,Z 355.255,A -85,B 0,C 180,E1 -24462.888,E2 -24462.888} C_VEL
LIN {X 0,Y 143.597,Z 355.224,A -85,B 0,C 180,E1 -24468.709,E2 -24468.709} C_VEL
LIN {X 0,Y 143.679,Z 355.21,A -85,B 0,C 180,E1 -24471.561,E2 -24471.561} C_VEL
LIN {X 0,Y 144.171,Z 355.15,A -85,B 0,C 180,E1 -24479.999,E2 -24479.999} C_VEL
LIN {X 0,Y 143.678,Z 355.21,A -85,B 0,C 180,E1 -24488.438,E2 -24488.438} C_VEL
LIN {X 0,Y 143.565,Z 355.222,A -85,B 0,C 180,E1 -24491.758,E2 -24491.758} C_VEL
LIN {X 0,Y 143.31,Z 355.256,A -85,B 0,C 180,E1 -24497.111,E2 -24497.111} C_VEL
LIN {X 0,Y 143.27,Z 355.261,A -85,B 0,C 180,E1 -24501.255,E2 -24501.255} C_VEL
LIN {X 0,Y 143.19,Z 355.268,A -85,B 0,C 180,E1 -24507.943,E2 -24507.943} C_VEL
LIN {X 0,Y 143.536,Z 355.39,A -85,B 0,C 180,E1 -24514.475,E2 -24514.475} C_VEL
LIN {X 0,Y 144.942,Z 361.741,A -85,B 0,C 180,E1 -24520.888,E2 -24520.888} C_VEL
LIN {X 0,Y 146.412,Z 367.079,A -85,B 0,C 180,E1 -24526.056,E2 -24526.056} C_VEL
LIN {X 0,Y 146.717,Z 368.998,A -85,B 0,C 180,E1 -24527.888,E2 -24527.888} C_VEL
LIN {X 0,Y 146.216,Z 371.491,A -85,B 0,C 180,E1 -24530.268,E2 -24530.268} C_VEL
LIN {X 0,Y 145.01,Z 375.624,A -85,B 0,C 180,E1 -24534.12,E2 -24534.12} C_VEL
LIN {X 0,Y 144.415,Z 394.861,A -85,B 0,C 180,E1 -24536.826,E2 -24536.826} C_VEL
LIN {X 0,Y 144.687,Z 410.129,A -85,B 0,C 180,E1 -24539.54,E2 -24539.54} C_VEL
LIN {X 0,Y 145.346,Z 424.332,A -85,B 0,C 180,E1 -24542.657,E2 -24542.657} C_VEL
LIN {X 0,Y 146.301,Z 438.408,A -85,B 0,C 180,E1 -24546.367,E2 -24546.367} C_VEL
LIN {X 0,Y 147.32,Z 448.255,A -85,B 0,C 180,E1 -24549.404,E2 -24549.404} C_VEL
LIN {X 0,Y 146.201,Z 458.167,A -85,B 0,C 180,E1 -24553.239,E2 -24553.239} C_VEL
LIN {X 0,Y 145.599,Z 467.206,A -85,B 0,C 180,E1 -24557.457,E2 -24557.457} C_VEL
LIN {X 0,Y 145.809,Z 475.894,A -85,B 0,C 180,E1 -24562.386,E2 -24562.386} C_VEL
LIN {X 0,Y 146.712,Z 482.751,A -85,B 0,C 180,E1 -24567.257,E2 -24567.257} C_VEL
LIN {X 0,Y 147.289,Z 485.85,A -85,B 0,C 180,E1 -24570.002,E2 -24570.002} C_VEL
LIN {X 0,Y 146.554,Z 487.933,A -85,B 0,C 180,E1 -24572.751,E2 -24572.751} C_VEL
LIN {X 0,Y 144.567,Z 490.582,A -85,B 0,C 180,E1 -24578.389,E2 -24578.389} C_VEL
LIN {X 0,Y 143.874,Z 492.127,A -85,B 0,C 180,E1 -24584.14,E2 -24584.14} C_VEL
LIN {X 0,Y 144.803,Z 492.814,A -85,B 0,C 180,E1 -24589.864,E2 -24589.864} C_VEL
LIN {X 0,Y 147.546,Z 492.687,A -85,B 0,C 180,E1 -24595.387,E2 -24595.387} C_VEL
LIN {X 0,Y 151.868,Z 491.859,A -85,B 0,C 180,E1 -24600.603,E2 -24600.603} C_VEL
LIN {X 0,Y 161.286,Z 489.276,A -85,B 0,C 180,E1 -24607.596,E2 -24607.596} C_VEL
LIN {X 0,Y 169.14,Z 486.673,A -85,B 0,C 180,E1 -24611.671,E2 -24611.671} C_VEL
LIN {X 0,Y 178.216,Z 483.461,A -85,B 0,C 180,E1 -24615.224,E2 -24615.224} C_VEL
LIN {X 0,Y 190.91,Z 478.15,A -85,B 0,C 180,E1 -24619.493,E2 -24619.493} C_VEL
LIN {X 0,Y 191.486,Z 477.655,A -85,B 0,C 180,E1 -24620.074,E2 -24620.074} C_VEL
LIN {X 0,Y 179.785,Z 477.846,A -85,B 0,C 180,E1 -24624.101,E2 -24624.101} C_VEL
LIN {X 0,Y 171.312,Z 477.011,A -85,B 0,C 180,E1 -24627.771,E2 -24627.771} C_VEL
LIN {X 0,Y 168.35,Z 476.439,A -85,B 0,C 180,E1 -24629.246,E2 -24629.246} C_VEL
LIN {X 0,Y 164.655,Z 475.784,A -85,B 0,C 180,E1 -24630.822,E2 -24630.822} C_VEL
LIN {X 0,Y 157.468,Z 474.462,A -85,B 0,C 180,E1 -24633.216,E2 -24633.216} C_VEL
LIN {X 0,Y 150.754,Z 472.516,A -85,B 0,C 180,E1 -24635.819,E2 -24635.819} C_VEL
LIN {X 0,Y 147.888,Z 470.965,A -85,B 0,C 180,E1 -24637.702,E2 -24637.702} C_VEL
LIN {X 0,Y 141.969,Z 465.068,A -85,B 0,C 180,E1 -24644.201,E2 -24644.201} C_VEL
LIN {X 0,Y 138.664,Z 459.084,A -85,B 0,C 180,E1 -24649.783,E2 -24649.783} C_VEL
LIN {X 0,Y 136.772,Z 451.872,A -85,B 0,C 180,E1 -24655.58,E2 -24655.58} C_VEL
LIN {X 0,Y 136.125,Z 444.405,A -85,B 0,C 180,E1 -24660.74,E2 -24660.74} C_VEL
LIN {X 0,Y 136.091,Z 434.23,A -85,B 0,C 180,E1 -24666.673,E2 -24666.673} C_VEL
LIN {X 0,Y 137.015,Z 425.303,A -85,B 0,C 180,E1 -24671.091,E2 -24671.091} C_VEL
LIN {X 0,Y 138.623,Z 413.034,A -85,B 0,C 180,E1 -24676.192,E2 -24676.192} C_VEL
LIN {X 0,Y 140.531,Z 400.422,A -85,B 0,C 180,E1 -24680.493,E2 -24680.493} C_VEL
LIN {X 0,Y 142.866,Z 386.735,A -85,B 0,C 180,E1 -24684.331,E2 -24684.331} C_VEL
LIN {X 0,Y 143.098,Z 383.847,A -85,B 0,C 180,E1 -24685.063,E2 -24685.063} C_VEL
LIN {X 0,Y 139.44,Z 369.573,A -85,B 0,C 180,E1 -24688.475,E2 -24688.475} C_VEL
LIN {X 0,Y 136.355,Z 356.703,A -85,B 0,C 180,E1 -24691.284,E2 -24691.284} C_VEL
LIN {X 0,Y 136.204,Z 356.163,A -85,B 0,C 180,E1 -24691.932,E2 -24691.932} C_VEL
LIN {X 0,Y 136.038,Z 356.163,A -85,B 0,C 180,E1 -24699.197,E2 -24699.197} C_VEL
LIN {X 0,Y 136.009,Z 356.165,A -85,B 0,C 180,E1 -24703.659,E2 -24703.659} C_VEL
LIN {X 0,Y 136.042,Z 356.162,A -85,B 0,C 180,E1 -24707.807,E2 -24707.807} C_VEL
LIN {X 0,Y 136.063,Z 356.159,A -85,B 0,C 180,E1 -24711.693,E2 -24711.693} C_VEL
LIN {X 0,Y 136.096,Z 356.154,A -85,B 0,C 180,E1 -24715.716,E2 -24715.716} C_VEL
LIN {X 0,Y 136.149,Z 356.145,A -85,B 0,C 180,E1 -24722.314,E2 -24722.314} C_VEL
LIN {X 0,Y 136.247,Z 356.135,A -85,B 0,C 180,E1 -24728.831,E2 -24728.831} C_VEL
LIN {X 0,Y 136.291,Z 356.132,A -85,B 0,C 180,E1 -24735.056,E2 -24735.056} C_VEL
LIN {X 0,Y 136.506,Z 356.101,A -85,B 0,C 180,E1 -24738.113,E2 -24738.113} C_VEL
LIN {X 0,Y 136.613,Z 356.089,A -85,B 0,C 180,E1 -24741.119,E2 -24741.119} C_VEL
LIN {X 0,Y 137.139,Z 356.026,A -85,B 0,C 180,E1 -24749.997,E2 -24749.997} C_VEL
LIN {X 0,Y 136.612,Z 356.091,A -85,B 0,C 180,E1 -24758.875,E2 -24758.875} C_VEL
LIN {X 0,Y 136.495,Z 356.106,A -85,B 0,C 180,E1 -24761.956,E2 -24761.956} C_VEL
LIN {X 0,Y 136.258,Z 356.137,A -85,B 0,C 180,E1 -24768.024,E2 -24768.024} C_VEL
LIN {X 0,Y 136.2,Z 356.141,A -85,B 0,C 180,E1 -24771.747,E2 -24771.747} C_VEL
LIN {X 0,Y 136.1,Z 356.156,A -85,B 0,C 180,E1 -24778.613,E2 -24778.613} C_VEL
LIN {X 0,Y 136.07,Z 356.158,A -85,B 0,C 180,E1 -24784.618,E2 -24784.618} C_VEL
LIN {X 0,Y 136.031,Z 356.161,A -85,B 0,C 180,E1 -24789.196,E2 -24789.196} C_VEL
LIN {X 0,Y 135.995,Z 356.169,A -85,B 0,C 180,E1 -24793.654,E2 -24793.654} C_VEL
LIN {X 0,Y 136.002,Z 356.165,A -85,B 0,C 180,E1 -24797.794,E2 -24797.794} C_VEL
LIN {X 0,Y 136.027,Z 356.164,A -85,B 0,C 180,E1 -24801.683,E2 -24801.683} C_VEL
LIN {X 0,Y 136.083,Z 356.156,A -85,B 0,C 180,E1 -24805.717,E2 -24805.717} C_VEL
LIN {X 0,Y 136.143,Z 356.151,A -85,B 0,C 180,E1 -24812.315,E2 -24812.315} C_VEL
LIN {X 0,Y 136.24,Z 356.139,A -85,B 0,C 180,E1 -24818.831,E2 -24818.831} C_VEL
LIN {X 0,Y 136.284,Z 356.128,A -85,B 0,C 180,E1 -24825.057,E2 -24825.057} C_VEL
LIN {X 0,Y 136.496,Z 356.107,A -85,B 0,C 180,E1 -24828.114,E2 -24828.114} C_VEL
